Yaskawa INFORM job: ariel_test_28-12.JBI

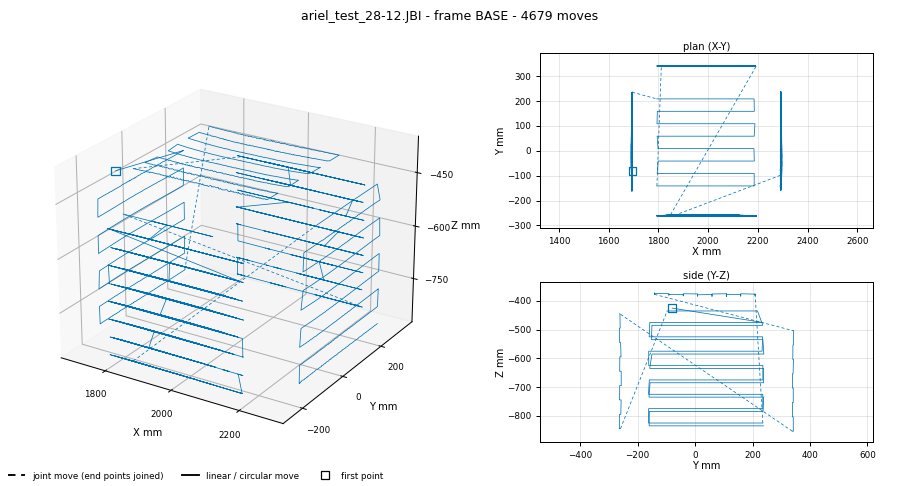
[picture p0: tool path of ariel_test_28-12.JBI in frame BASE, 4679 of 4679 moves have a stored position in this frame; points joined in program order, loops and branches not executed]
/JOB
//NAME ARIEL_TEST
//POS
///NPOS 4679,0,0,0,0,0
///TOOL 0
///POSTYPE BASE
///RECTAN
///RCONF 1,0,0,0,0,0,0,0,0,0,0,0,0,0,0,0,0,0,0,0,0,0,0,0
C00000=1696.132000,-80.047400,-425.128800,-2.796034,72.857313,-92.928025
C00001=1694.988400,235.674100,-475.128800,91.633140,81.554813,1.615741
C00002=1694.763900,232.398000,-475.128800,113.107598,87.891726,23.090199
C00003=1694.793600,228.055300,-475.128800,-70.657155,88.596464,-160.663095
C00004=1695.151200,224.781200,-475.128800,-66.440186,88.699596,-156.446126
C00005=1695.130800,221.009900,-475.128800,-43.934404,88.980346,-133.934614
C00006=1695.054300,219.997000,-475.128800,-8.926682,88.791270,-98.926893
C00007=1695.058500,217.094900,-475.128800,-159.081732,88.567816,110.924629
C00008=1694.887700,215.803300,-475.128800,-11.676880,88.842836,-101.677090
C00009=1695.188800,212.462700,-475.128800,-4.371668,86.453602,-94.377608
C00010=1695.133100,208.131800,-475.128800,-42.633790,89.398605,-132.634000
C00011=1695.189200,206.048000,-475.128800,-13.493156,89.587681,-103.493367
C00012=1695.116300,201.470900,-475.128800,50.191103,88.590734,-39.803378
C00013=1694.965700,197.460000,-475.128800,48.460770,89.272554,-41.539440
C00014=1695.140400,191.185200,-475.128800,17.492401,89.639247,-72.502079
C00015=1694.918000,187.331000,-475.128800,31.885101,88.860024,-58.109380
C00016=1695.110400,184.389700,-475.128800,64.853093,89.364227,-25.147118
C00017=1694.969600,179.240300,-475.128800,-12.100869,87.914644,-102.106809
C00018=1695.056000,175.417900,-475.128800,38.898105,88.590734,-51.090647
C00019=1694.747200,170.987700,-475.128800,47.629982,87.817241,-42.347311
C00020=1694.650000,164.775100,-475.128800,16.432430,88.510520,-73.562051
C00021=1694.533900,162.575300,-475.128800,42.089480,88.390199,-47.899272
C00022=1694.373600,158.045800,-475.128800,56.997841,88.556357,-32.990910
C00023=1695.089100,155.989400,-475.128800,-6.348372,88.344362,-96.354312
C00024=1695.185800,152.477800,-475.128800,-65.809932,88.149557,-155.821602
C00025=1694.724600,149.203700,-475.128800,6.033246,87.261472,-83.961235
C00026=1695.104800,146.728300,-475.128800,19.486295,88.923050,-70.513916
C00027=1694.834300,143.853900,-475.128800,47.733114,88.705326,-42.255637
C00028=1693.934200,141.094100,-475.128800,115.748934,87.490655,25.725805
C00029=1693.799200,137.257000,-475.128800,99.190453,86.671326,9.173054
C00030=1693.895200,133.651800,-475.128800,38.038668,87.828700,-51.938624
C00031=1693.476900,130.746700,-475.128800,21.720830,87.026560,-68.250733
C00032=1694.334900,128.603600,-475.128800,25.382030,86.785917,-64.583803
C00033=1695.164800,125.432200,-475.128800,143.904080,88.711055,53.898140
C00034=1694.863300,121.656100,-475.128800,8.382373,87.026560,-81.606379
C00035=1693.391000,117.740300,-475.128800,20.064982,87.748486,-69.923769
C00036=1694.429700,115.474900,-475.128800,6.205133,87.381793,-83.789348
C00037=1693.264100,112.358400,-475.128800,47.624252,88.350092,-42.364499
C00038=1694.551300,109.480100,-475.128800,-7.053110,87.507844,-97.059050
C00039=1694.104100,106.646300,-475.128800,8.141730,87.198447,-81.847021
C00040=1693.197200,102.981000,-475.128800,-2.950733,87.444819,-92.950943
C00041=1694.004100,100.489400,-475.128800,16.031359,86.929157,-73.951663
C00042=1694.629400,96.503800,-475.128800,0.435448,86.785917,-89.559033
C00043=1693.339800,94.279400,-475.128800,4.153944,86.602571,-85.840537
C00044=1693.243600,89.591100,-475.128800,30.068825,88.395929,-59.919926
C00045=1694.046600,86.533600,-475.128800,-0.435448,87.101044,-90.435658
C00046=1694.079400,83.430500,-475.128800,-14.896903,86.636948,-104.920031
C00047=1694.640600,81.259500,-475.128800,-7.591691,81.062069,-97.683574
C00048=1693.579900,77.591900,-475.128800,-3.701307,86.728621,-93.707247
C00049=1694.579600,74.118800,-475.128800,8.061516,86.677055,-81.927235
C00050=1694.602200,71.620100,-475.128800,5.655093,86.379117,-84.333658
C00051=1693.230300,67.936100,-475.128800,7.574502,86.682785,-82.408520
C00052=1692.692500,63.461100,-475.128800,3.368992,87.301579,-86.625489
C00053=1693.515800,60.204800,-475.128800,-3.540879,86.751540,-93.541090
C00054=1694.397600,57.070500,-475.128800,-1.867842,86.321821,-91.873782
C00055=1695.083600,51.313600,-475.128800,-46.077266,88.854295,-136.083206
C00056=1693.552700,49.260100,-475.128800,3.449206,86.327551,-86.545275
C00057=1693.236600,43.220200,-475.128800,-9.150136,86.361928,-99.167535
C00058=1692.438400,40.123200,-475.128800,-10.250215,86.860402,-100.267614
C00059=1693.005200,36.124700,-475.128800,-0.458366,86.281714,-90.458577
C00060=1694.308400,31.082800,-475.128800,-2.051189,86.493709,-92.057129
C00061=1692.704700,27.503400,-475.128800,2.784575,87.782864,-87.209906
C00062=1693.177400,25.817900,-475.128800,10.880469,87.307309,-79.108283
C00063=1692.952200,22.582800,-475.128800,5.826981,86.052531,-84.161771
C00064=1693.146000,20.159200,-475.128800,3.770062,88.063613,-86.224419
C00065=1694.605100,16.625400,-475.128800,-10.141353,85.754593,-100.170211
C00066=1693.774400,12.699800,-475.128800,-8.978249,86.957805,-98.989918
C00067=1694.221300,10.877900,-475.128800,9.396508,85.456655,-80.569325
C00068=1693.353500,8.692400,-475.128800,-10.588260,87.479196,-100.599930
C00069=1695.395900,6.553600,-475.128800,-14.278108,75.962744,-104.696578
C00070=1694.514400,2.859000,-475.128800,-3.775792,86.293174,-93.781732
C00071=1694.492400,-1.569500,-475.128800,-24.327788,87.284391,-114.356646
C00072=1692.776900,-3.735100,-475.128800,-27.318628,87.261472,-117.347486
C00073=1694.690400,-6.961900,-475.128800,-12.060762,85.788971,-102.089620
C00074=1694.113600,-9.973800,-475.128800,-4.881600,87.410441,-94.887540
C00075=1695.315300,-12.616400,-475.128800,5.523313,88.338633,-84.471168
C00076=1693.186800,-16.477300,-475.128800,-14.810959,86.969264,-104.828358
C00077=1694.776500,-17.860800,-475.128800,-8.147460,86.396306,-98.159129
C00078=1693.169700,-22.210600,-475.128800,-23.491270,87.536492,-113.508669
C00079=1694.236600,-24.585300,-475.128800,-9.763201,86.023883,-99.786330
C00080=1693.849200,-28.361700,-475.128800,-19.784233,87.204176,-109.807361
C00081=1694.081800,-32.852400,-475.128800,-27.788453,87.393252,-117.817311
C00082=1694.169000,-36.280800,-475.128800,-40.880539,87.215636,-130.915127
C00083=1694.436000,-38.893400,-475.128800,-11.493533,86.333281,-101.516662
C00084=1693.377800,-42.844200,-475.128800,-15.429753,87.020830,-105.452882
C00085=1693.729500,-46.013500,-475.128800,-5.689471,87.284391,-95.695411
C00086=1693.512300,-48.882800,-475.128800,-21.319760,87.272931,-111.337159
C00087=1694.121900,-53.479200,-475.128800,-2.097026,87.370334,-92.097236
C00088=1694.254700,-55.606600,-475.128800,-8.663122,87.123962,-98.674791
C00089=1695.480200,-60.498300,-475.128800,-7.551584,88.361551,-97.551794
C00090=1694.880500,-63.263300,-475.128800,-10.066868,86.344740,-100.089997
C00091=1695.519400,-67.371500,-475.128800,-4.279995,86.465061,-94.291664
C00092=1695.154700,-69.634000,-475.128800,-16.690261,86.906238,-106.713389
C00093=1694.837500,-73.212500,-475.128800,-14.346863,87.209906,-104.364262
C00094=1695.406500,-77.363100,-475.128800,-22.505782,86.992182,-112.534641
C00095=1695.106600,-81.047500,-475.128800,-14.696367,88.143827,-104.702307
C00096=1694.416400,-84.097200,-475.128800,-20.317083,87.628165,-110.334483
C00097=1695.519600,-87.829700,-475.128800,82.540300,88.986075,-7.459910
C00098=1694.707800,-90.627800,-475.128800,-9.660068,86.911968,-99.671738
C00099=1695.330000,-93.501100,-475.128800,-21.336948,87.679731,-111.354347
C00100=1695.363400,-99.305300,-475.128800,-13.200948,87.582329,-103.212617
C00101=1694.622800,-103.431100,-475.128800,-32.750268,88.315715,-122.761937
C00102=1695.475000,-107.547000,-475.128800,2.710090,87.840160,-87.290120
C00103=1694.908200,-111.406000,-475.128800,-12.536317,88.235500,-102.542257
C00104=1695.600100,-115.157400,-475.128800,63.403510,89.793946,-26.596701
C00105=1694.895300,-121.393400,-475.128800,-19.469106,88.373010,-109.475046
C00106=1695.267600,-125.384400,-475.128800,-1.890761,88.424577,-91.896701
C00107=1694.736800,-129.294900,-475.128800,-21.904177,89.049101,-111.910117
C00108=1694.843800,-133.799800,-475.128800,-11.694069,88.355822,-101.694279
C00109=1695.271400,-139.102900,-475.128800,-14.432807,88.751162,-104.438747
C00110=1695.095400,-144.244300,-475.128800,-2.475178,88.281337,-92.475388
C00111=1694.850400,-148.261100,-475.128800,-17.985145,88.453224,-107.991085
C00112=1695.327400,-150.030400,-475.128800,46.959621,88.785540,-43.034860
C00113=1695.394800,-153.452400,-475.128800,127.414354,87.192717,37.385496
C00114=1694.805400,-157.684500,-475.128800,-67.276704,86.963534,-157.305563
C00115=1694.500400,-159.876400,-525.128800,-78.924936,82.712187,-169.011090
C00116=1694.421900,-156.702300,-525.128800,-95.036509,88.539168,174.964122
C00117=1694.689000,-153.571800,-525.128800,-16.822041,89.484548,-106.822251
C00118=1694.622100,-150.053500,-525.128800,-18.987821,88.865754,-108.993761
C00119=1694.362400,-147.366300,-525.128800,-40.221637,88.865754,-130.221848
C00120=1694.470800,-144.581100,-525.128800,-53.118917,88.842836,-143.124857
C00121=1694.487200,-142.921900,-525.128800,-69.241950,88.911591,-159.247890
C00122=1694.727000,-138.966100,-525.128800,-58.361481,89.238177,-148.367421
C00123=1694.454100,-135.239700,-525.128800,-40.026832,88.573546,-130.032772
C00124=1694.239400,-130.327700,-525.128800,-74.828288,88.739703,-164.834228
C00125=1694.291700,-126.172900,-525.128800,-35.735378,88.327174,-125.747047
C00126=1693.961600,-120.293700,-525.128800,-44.455795,88.161016,-134.467465
C00127=1694.229600,-117.327700,-525.128800,-39.677327,88.378740,-129.688997
C00128=1693.955300,-112.124600,-525.128800,-39.012696,88.550627,-129.018636
C00129=1694.120500,-109.056600,-525.128800,-37.087558,88.544898,-127.099228
C00130=1693.350900,-104.310500,-525.128800,-49.807221,87.840160,-139.824620
C00131=1693.551400,-100.440500,-525.128800,-37.339660,87.800053,-127.357059
C00132=1693.489700,-95.539000,-525.128800,-61.277836,87.232824,-151.306695
C00133=1693.865700,-92.922100,-525.128800,-39.562736,87.439089,-129.591594
C00134=1693.249200,-88.499300,-525.128800,-41.917592,88.774081,-131.923532
C00135=1693.006200,-86.270900,-525.128800,-63.541019,88.373010,-153.546960
C00136=1693.393100,-79.718400,-525.128800,-36.887023,87.857348,-126.904422
C00137=1693.031700,-76.883500,-525.128800,-29.226577,87.651083,-119.249706
C00138=1693.235600,-73.650000,-525.128800,-33.667000,87.943292,-123.684399
C00139=1692.490700,-67.602900,-525.128800,-23.044363,87.496385,-113.061762
C00140=1693.098200,-63.993300,-525.128800,-33.162797,87.502114,-123.191656
C00141=1692.056100,-60.055400,-525.128800,-46.856488,88.653760,-136.862429
C00142=1692.699200,-57.465500,-525.128800,-34.411845,88.172475,-124.423515
C00143=1692.339800,-53.601900,-525.128800,-27.215495,88.034965,-117.227165
C00144=1692.501500,-49.582900,-525.128800,-18.157033,88.092261,-108.168702
C00145=1691.991300,-47.866600,-525.128800,-46.999728,88.292796,-137.017127
C00146=1692.189200,-44.341200,-525.128800,-17.383540,87.759945,-107.395209
C00147=1691.755300,-40.515100,-525.128800,-28.390059,88.464684,-118.401728
C00148=1692.760800,-37.856600,-525.128800,-26.757129,86.321821,-116.803176
C00149=1692.377400,-34.007100,-525.128800,-22.929771,88.831377,-112.929981
C00150=1692.333500,-29.550300,-525.128800,-22.843827,88.355822,-112.849767
C00151=1691.906200,-26.667400,-525.128800,-25.783101,88.212582,-115.794770
C00152=1692.601600,-23.052500,-525.128800,-46.506984,87.651083,-136.530113
C00153=1691.715700,-19.895400,-525.128800,-46.524173,88.378740,-136.535843
C00154=1691.346100,-17.017200,-525.128800,-23.370948,88.269878,-113.382618
C00155=1691.553100,-15.002600,-525.128800,-34.423304,88.350092,-124.434974
C00156=1691.985700,-9.968700,-525.128800,-10.416373,88.075072,-100.422313
C00157=1691.467400,-6.304400,-525.128800,-5.809792,88.023506,-95.815732
C00158=1691.911100,-3.077000,-525.128800,-20.746802,88.716785,-110.752742
C00159=1691.862600,0.698400,-525.128800,-8.072975,88.052154,-98.078915
C00160=1691.612400,3.808600,-525.128800,-39.127288,89.049101,-129.127498
C00161=1692.269100,7.928600,-525.128800,-24.430920,87.204176,-114.454049
C00162=1691.326600,9.877800,-525.128800,-26.018013,88.928779,-116.023954
C00163=1691.066200,12.948400,-525.128800,-66.268299,87.828700,-156.279968
C00164=1691.291700,15.880200,-525.128800,-9.734553,87.519303,-99.746223
C00165=1691.603000,21.223400,-525.128800,-14.014548,88.659489,-104.020488
C00166=1691.244300,23.875200,-525.128800,20.116548,88.728244,-69.877933
C00167=1691.672000,27.568300,-525.128800,-40.141423,88.258419,-130.153093
C00168=1691.918800,29.995600,-525.128800,-5.030569,87.295850,-95.036509
C00169=1691.532200,34.742900,-525.128800,62.280512,89.272554,-27.713969
C00170=1691.777300,36.968100,-525.128800,1.638659,87.633895,-88.361551
C00171=1692.094100,41.761800,-525.128800,7.465640,88.842836,-82.528841
C00172=1692.187100,44.735300,-525.128800,16.243353,87.937562,-73.745398
C00173=1691.171000,47.416500,-525.128800,33.867535,88.968886,-56.132675
C00174=1691.446100,51.083700,-525.128800,10.582530,88.504791,-79.417680
C00175=1691.301500,52.729200,-525.128800,50.815627,89.163692,-39.178854
C00176=1691.411400,56.907700,-525.128800,101.276020,88.808458,11.270080
C00177=1691.256200,60.771300,-525.128800,20.420216,88.487602,-69.574265
C00178=1691.909500,62.038600,-525.128800,2.807493,88.390199,-87.192717
C00179=1692.124100,67.281200,-525.128800,17.062683,88.350092,-72.931798
C00180=1692.099300,70.838300,-525.128800,26.373247,88.441765,-63.615504
C00181=1692.157500,72.684000,-525.128800,18.649776,88.378740,-71.338975
C00182=1691.565800,76.598500,-525.128800,3.036676,88.464684,-86.963534
C00183=1691.909400,80.224700,-525.128800,105.017434,89.123585,15.017224
C00184=1692.286100,84.108200,-525.128800,18.718531,88.298526,-71.275950
C00185=1691.948700,86.578200,-525.128800,38.038668,88.430306,-51.950083
C00186=1691.934400,90.287100,-525.128800,18.030982,88.607923,-71.963499
C00187=1692.085000,93.239200,-525.128800,42.868702,88.040695,-47.114319
C00188=1692.449200,96.809000,-525.128800,-8.600097,87.565140,-98.611766
C00189=1691.972100,100.726900,-525.128800,51.932895,88.327174,-38.055857
C00190=1692.777100,102.244500,-525.128800,51.503176,87.003641,-38.456927
C00191=1692.585200,107.563200,-525.128800,43.831271,88.052154,-46.151750
C00192=1692.245700,109.667000,-525.128800,90.315337,88.562086,0.315127
C00193=1692.710700,113.138300,-525.128800,77.658700,88.017776,-12.330052
C00194=1692.487800,115.926400,-525.128800,54.436720,88.441765,-35.552031
C00195=1692.585500,119.868600,-525.128800,70.542564,88.550627,-19.451917
C00196=1692.703700,124.136900,-525.128800,68.038738,87.857348,-21.950013
C00197=1693.348100,127.989000,-525.128800,14.123410,89.008993,-75.871071
C00198=1693.014600,131.500300,-525.128800,52.689199,87.960481,-37.293823
C00199=1693.004100,135.286200,-525.128800,69.190383,88.023506,-20.798368
C00200=1693.062300,138.337900,-525.128800,70.296192,88.670948,-19.698289
C00201=1693.695300,142.853900,-525.128800,36.308335,87.164069,-53.657498
C00202=1693.927400,146.038400,-525.128800,25.032526,87.926103,-64.956225
C00203=1693.303900,150.565200,-525.128800,86.190041,88.590734,-3.810169
C00204=1693.469800,156.957300,-525.128800,171.486268,89.662165,81.486058
C00205=1693.614100,160.194900,-525.128800,68.479916,88.057884,-21.508836
C00206=1693.876900,164.625000,-525.128800,83.050232,88.745433,-6.949978
C00207=1694.292400,168.627500,-525.128800,69.012766,88.831377,-20.987444
C00208=1693.978700,172.496500,-525.128800,66.422997,88.390199,-23.565754
C00209=1694.116300,176.139200,-525.128800,93.793191,88.991805,3.792981
C00210=1694.081500,181.483900,-525.128800,58.418777,88.550627,-31.569975
C00211=1694.426900,184.221100,-525.128800,61.741932,88.648030,-28.252549
C00212=1694.402500,190.301700,-525.128800,32.217417,89.008993,-57.777064
C00213=1694.649600,195.955200,-525.128800,59.765228,88.722515,-30.229253
C00214=1694.804700,197.877500,-525.128800,52.637633,89.026182,-37.356848
C00215=1694.710300,202.217900,-525.128800,65.454699,89.324120,-24.545512
C00216=1694.828100,206.371000,-525.128800,47.612793,89.014723,-42.381688
C00217=1694.680600,209.763000,-525.128800,130.336439,88.579275,40.324770
C00218=1694.784900,212.216100,-525.128800,55.021137,88.917320,-34.979073
C00219=1694.849000,214.324600,-525.128800,1.747521,87.880267,-88.252689
C00220=1694.724400,215.988100,-525.128800,31.403817,88.481872,-58.584935
C00221=1694.889400,219.187200,-525.128800,4.898789,88.745433,-85.101421
C00222=1694.788600,221.768000,-525.128800,-122.830692,84.247714,147.301720
C00223=1694.756300,224.941700,-525.128800,-136.604598,88.269878,133.407493
C00224=1694.729100,227.663700,-525.128800,7.081758,89.822594,-82.918452
C00225=1694.687300,230.259700,-525.128800,50.511959,89.135044,-39.488251
C00226=1694.723200,234.923700,-525.128800,92.355067,83.353900,2.337668
C00227=1694.806300,233.203100,-575.128800,103.653795,82.620514,13.544722
C00228=1694.742300,231.059300,-575.128800,75.120497,86.952075,-14.862525
C00229=1694.693700,226.262900,-575.128800,-78.369167,89.008993,-168.369378
C00230=1694.887000,224.564300,-575.128800,-9.866333,89.862701,-99.866544
C00231=1694.695600,221.286200,-575.128800,-22.906853,89.478819,-112.907063
C00232=1694.713100,219.344300,-575.128800,73.464648,89.387146,-16.535562
C00233=1694.584600,216.524100,-575.128800,139.297499,89.725191,49.297289
C00234=1694.630300,213.463400,-575.128800,27.129552,88.968886,-62.870659
C00235=1694.668100,210.962700,-575.128800,162.061112,88.728244,72.055172
C00236=1694.607400,208.721700,-575.128800,108.357778,89.049101,18.357568
C00237=1694.629100,206.423000,-575.128800,24.935123,89.094937,-65.065087
C00238=1694.628700,202.253300,-575.128800,69.952417,89.220988,-20.042064
C00239=1694.515400,199.405300,-575.128800,104.089243,89.112126,14.083303
C00240=1694.346400,194.510600,-575.128800,53.239238,88.791270,-36.755243
C00241=1694.248400,188.122200,-575.128800,78.437922,88.527709,-11.556559
C00242=1694.228200,183.278500,-575.128800,96.904352,88.224041,6.904141
C00243=1693.970700,179.423000,-575.128800,78.953584,88.218312,-11.040897
C00244=1693.868200,172.668500,-575.128800,53.353830,88.579275,-36.640651
C00245=1693.812400,169.950500,-575.128800,112.523181,88.367281,22.517241
C00246=1693.709200,166.789600,-575.128800,79.956260,89.106396,-10.038221
C00247=1693.646200,162.728400,-575.128800,71.470755,88.212582,-18.517996
C00248=1693.661500,159.420200,-575.128800,85.055585,88.206853,-4.938896
C00249=1693.425500,155.227500,-575.128800,91.696166,88.034965,1.695955
C00250=1693.320300,151.517000,-575.128800,78.861911,88.648030,-11.132570
C00251=1693.201800,147.367900,-575.128800,74.587646,88.390199,-15.406835
C00252=1692.996500,142.122500,-575.128800,106.043029,87.496385,16.031359
C00253=1692.897500,140.572100,-575.128800,57.874467,88.109450,-32.114284
C00254=1692.852900,136.432100,-575.128800,102.232859,86.997912,12.215460
C00255=1692.607500,133.096600,-575.128800,108.311942,88.166746,18.300272
C00256=1692.506800,127.929600,-575.128800,84.007072,88.097991,-5.987409
C00257=1692.637100,126.345400,-575.128800,103.814223,88.487602,13.808283
C00258=1692.460100,120.405100,-575.128800,121.426946,87.891726,31.409546
C00259=1692.265600,116.228300,-575.128800,86.465061,88.636571,-3.535150
C00260=1692.250600,112.447400,-575.128800,102.278696,88.510520,12.272756
C00261=1692.136600,109.594700,-575.128800,72.055172,88.413117,-17.933579
C00262=1691.893000,104.059400,-575.128800,56.694174,88.476143,-33.294577
C00263=1691.813200,101.461400,-575.128800,106.782144,88.636571,16.781934
C00264=1691.820100,97.498400,-575.128800,48.300342,88.716785,-41.694139
C00265=1691.695000,93.109800,-575.128800,97.007484,88.642300,7.007274
C00266=1691.744500,90.048900,-575.128800,96.686628,88.670948,6.686417
C00267=1691.683500,85.860600,-575.128800,134.988857,88.602193,44.982916
C00268=1691.585900,83.286900,-575.128800,85.640002,89.364227,-4.360209
C00269=1691.337700,79.352400,-575.128800,57.043678,88.728244,-32.950803
C00270=1691.369100,74.414100,-575.128800,75.424164,89.255365,-14.576046
C00271=1691.218900,72.542400,-575.128800,119.862771,89.610599,29.862560
C00272=1691.295600,67.757100,-575.128800,66.852716,89.106396,-23.147495
C00273=1691.304300,64.282100,-575.128800,163.579451,87.828700,73.567781
C00274=1691.097900,62.191800,-575.128800,56.992112,89.152233,-33.002369
C00275=1690.987500,56.823900,-575.128800,-140.225691,89.284013,129.774941
C00276=1691.165600,55.524500,-575.128800,34.383197,88.367281,-55.605554
C00277=1691.027500,51.901500,-575.128800,118.229841,89.725191,28.229631
C00278=1690.928900,47.456300,-575.128800,56.241537,88.653760,-33.747214
C00279=1690.984000,45.810200,-575.128800,-8.462587,88.298526,-98.468527
C00280=1691.087500,41.819000,-575.128800,-52.030297,89.146503,-142.036237
C00281=1691.043600,39.213400,-575.128800,142.305528,89.513196,52.305317
C00282=1691.026500,35.327600,-575.128800,-28.487462,89.564763,-118.487672
C00283=1690.873600,32.032400,-575.128800,45.848083,89.180881,-44.152128
C00284=1690.821200,30.213600,-575.128800,33.913372,88.161016,-56.069650
C00285=1690.929400,26.425500,-575.128800,-12.662367,88.613653,-102.668307
C00286=1690.815600,23.772000,-575.128800,-111.904387,89.335579,158.096244
C00287=1690.808600,19.852900,-575.128800,57.759875,89.610599,-32.240335
C00288=1690.950900,16.612700,-575.128800,-115.525480,89.856971,154.475151
C00289=1690.737500,11.905700,-575.128800,-109.039598,88.894402,160.966763
C00290=1690.920900,8.527600,-575.128800,-84.270633,89.026182,-174.270843
C00291=1690.739300,5.954200,-575.128800,167.045845,89.885619,77.045635
C00292=1690.841100,2.739900,-575.128800,-19.812881,89.627788,-109.813091
C00293=1690.672400,-1.372900,-575.128800,31.770510,89.581951,-58.229701
C00294=1690.806600,-3.662500,-575.128800,-41.470685,88.464684,-131.476625
C00295=1691.056800,-8.688600,-575.128800,-28.029095,89.049101,-118.029306
C00296=1690.987500,-12.668800,-575.128800,6.514530,88.814188,-83.485680
C00297=1690.795700,-20.036900,-575.128800,-41.344634,89.432982,-131.344845
C00298=1690.997900,-24.547800,-575.128800,-76.890936,89.049101,-166.896876
C00299=1690.918100,-30.269200,-575.128800,-25.966447,89.135044,-115.972387
C00300=1691.294200,-35.152800,-575.128800,-25.296087,88.224041,-115.302027
C00301=1691.022000,-39.070400,-575.128800,-46.294990,89.037641,-136.300930
C00302=1691.086400,-41.699200,-575.128800,-46.799193,88.762622,-136.805133
C00303=1691.265600,-47.309800,-575.128800,-46.346556,88.848565,-136.352496
C00304=1691.355200,-50.600100,-575.128800,-19.864447,88.991805,-109.864657
C00305=1691.892600,-55.259700,-575.128800,-41.751435,88.075072,-131.763104
C00306=1691.475100,-59.480400,-575.128800,-78.111336,88.178205,-168.117276
C00307=1691.274300,-63.897400,-575.128800,-78.472300,88.212582,-168.478240
C00308=1691.851500,-66.924200,-575.128800,-38.823620,87.966210,-128.841019
C00309=1691.543400,-71.041500,-575.128800,-128.193577,87.800053,141.829973
C00310=1691.724300,-73.351300,-575.128800,-3.111161,88.029236,-93.111371
C00311=1692.211900,-78.850500,-575.128800,-89.123585,88.877213,-179.123795
C00312=1692.125800,-79.622100,-575.128800,-76.782074,88.837106,-166.788014
C00313=1692.001400,-84.001300,-575.128800,-76.438299,88.648030,-166.438510
C00314=1692.577700,-87.866400,-575.128800,-56.258726,88.825647,-146.258936
C00315=1692.045800,-91.980500,-575.128800,-95.620926,88.579275,174.379705
C00316=1692.173600,-94.043900,-575.128800,-85.508221,87.777134,-175.508432
C00317=1692.553100,-100.118900,-575.128800,-73.298491,88.109450,-163.304431
C00318=1692.848000,-103.049700,-575.128800,-65.809932,88.143827,-155.821602
C00319=1693.065100,-107.930200,-575.128800,-76.151821,87.513574,-166.163490
C00320=1692.948700,-112.113100,-575.128800,-59.564692,88.733974,-149.570632
C00321=1693.011800,-116.306100,-575.128800,-82.815320,88.000588,-172.815530
C00322=1693.309500,-121.879900,-575.128800,-72.765640,87.055207,-162.788769
C00323=1693.330000,-125.985400,-575.128800,-81.228227,87.410441,-171.234167
C00324=1693.636700,-128.998600,-575.128800,-81.950153,88.052154,-171.950364
C00325=1693.762900,-132.765600,-575.128800,-79.560919,88.304255,-169.566859
C00326=1693.867800,-137.386300,-575.128800,-126.560647,88.648030,143.445714
C00327=1694.041100,-140.149600,-575.128800,-69.791989,88.069343,-159.803659
C00328=1694.038600,-142.787500,-575.128800,-94.813056,88.057884,175.187575
C00329=1694.000600,-144.618300,-575.128800,-71.533781,87.966210,-161.545450
C00330=1694.203100,-147.692000,-575.128800,-95.334448,88.573546,174.666184
C00331=1694.311200,-152.225200,-575.128800,-102.175564,89.255365,167.825068
C00332=1694.376400,-154.259400,-575.128800,31.060042,89.719461,-58.940168
C00333=1694.414700,-156.252300,-575.128800,-114.247784,87.341686,155.775765
C00334=1694.517600,-158.357200,-575.128800,-103.183969,88.888672,166.822392
C00335=1694.945200,-161.433200,-575.128800,-94.738571,78.260305,175.359463
C00336=1694.553400,-161.479100,-625.128800,-68.806502,79.050987,-159.156216
C00337=1694.756200,-158.430600,-625.128800,-76.220575,83.760700,-166.301000
C00338=1694.559700,-156.743200,-625.128800,-104.387181,86.413495,165.636369
C00339=1694.303200,-153.567800,-625.128800,-61.564315,87.559410,-151.587444
C00340=1694.320200,-150.343100,-625.128800,-84.299280,87.450548,-174.299491
C00341=1693.989800,-147.719700,-625.128800,-78.013933,86.992182,-168.031333
C00342=1693.810300,-142.914800,-625.128800,-75.481460,87.101044,-165.498859
C00343=1693.818300,-139.261400,-625.128800,-95.110994,87.370334,174.895367
C00344=1693.699800,-134.943000,-625.128800,-92.120154,88.023506,177.880477
C00345=1693.573700,-130.480400,-625.128800,-96.119400,87.645354,173.886961
C00346=1693.153700,-126.406300,-625.128800,-86.946345,87.123962,-176.952285
C00347=1693.106600,-121.856200,-625.128800,-78.718671,87.095314,-168.730341
C00348=1692.960600,-118.089600,-625.128800,-84.133123,87.926103,-174.139063
C00349=1692.713100,-112.713100,-625.128800,-82.248091,87.971940,-172.254032
C00350=1692.412300,-110.341100,-625.128800,-74.702237,88.246960,-164.708177
C00351=1692.432900,-106.464300,-625.128800,-76.358085,88.212582,-166.364025
C00352=1692.347100,-102.865600,-625.128800,-97.574713,88.046424,172.431648
C00353=1692.024000,-98.807000,-625.128800,-67.660586,87.725568,-157.677985
C00354=1692.063300,-93.005100,-625.128800,-73.859989,88.860024,-163.860200
C00355=1692.032700,-88.429400,-625.128800,-83.353900,87.954751,-173.354110
C00356=1691.922900,-85.154300,-625.128800,-81.577731,87.897455,-171.583671
C00357=1691.639900,-80.293400,-625.128800,-118.332973,88.103720,151.679117
C00358=1691.561900,-76.884200,-625.128800,-63.225893,88.499061,-153.237562
C00359=1691.419600,-71.985100,-625.128800,-22.769343,86.459331,-112.809660
C00360=1691.352000,-67.828900,-625.128800,-54.316399,88.796999,-144.322339
C00361=1691.103500,-64.509200,-625.128800,-48.231587,88.373010,-138.237527
C00362=1691.180500,-61.617600,-625.128800,-24.001202,88.997534,-114.001412
C00363=1691.089200,-57.626000,-625.128800,-73.819882,88.928779,-163.820093
C00364=1691.159300,-54.104900,-625.128800,151.656199,89.925726,61.655988
C00365=1691.154800,-50.557900,-625.128800,-38.674651,89.020453,-128.674862
C00366=1691.026100,-48.692300,-625.128800,-45.722032,88.665219,-135.727972
C00367=1690.951200,-44.611100,-625.128800,-74.421488,89.014723,-164.421698
C00368=1690.795700,-42.130000,-625.128800,-39.333553,88.957427,-129.333763
C00369=1690.759500,-37.278500,-625.128800,-49.532201,89.467360,-139.532412
C00370=1690.847700,-34.944000,-625.128800,-94.371878,89.369957,175.628753
C00371=1690.742800,-31.427000,-625.128800,-121.129007,89.455901,148.871624
C00372=1690.778000,-28.339400,-625.128800,-12.278486,89.020453,-102.278696
C00373=1690.609300,-25.061600,-625.128800,40.049750,89.748109,-49.944731
C00374=1690.613800,-21.692600,-625.128800,124.732912,89.043371,34.726972
C00375=1690.768600,-19.120600,-625.128800,-153.718847,88.756892,116.287514
C00376=1690.638900,-13.464400,-625.128800,-174.746398,89.031912,95.254233
C00377=1690.663300,-8.718300,-625.128800,151.908300,89.536115,61.908090
C00378=1690.737200,-6.140600,-625.128800,-21.663534,89.352768,-111.663745
C00379=1690.630500,-4.212800,-625.128800,-49.566579,89.324120,-139.566789
C00380=1690.744500,-0.158000,-625.128800,-167.389620,88.934509,102.611012
C00381=1690.633000,2.934700,-625.128800,54.889357,88.900131,-35.105124
C00382=1690.812700,6.829400,-625.128800,19.423269,89.444441,-70.576941
C00383=1690.813200,11.135600,-625.128800,109.589637,89.484548,19.589427
C00384=1690.874600,15.819000,-625.128800,-149.209669,89.450171,120.796692
C00385=1691.095200,20.063900,-625.128800,104.009029,88.017776,14.003089
C00386=1690.840000,22.530800,-625.128800,95.655304,89.329850,5.655093
C00387=1690.961700,26.623700,-625.128800,68.869527,88.791270,-21.124954
C00388=1690.939700,30.121100,-625.128800,56.751470,89.392875,-33.248741
C00389=1690.878700,33.744200,-625.128800,40.215908,88.923050,-49.784303
C00390=1690.938300,36.801700,-625.128800,175.405299,89.496008,85.405089
C00391=1690.897900,40.528300,-625.128800,-120.212275,89.897078,149.782627
C00392=1691.261800,42.787500,-625.128800,84.958182,88.882943,-5.042029
C00393=1691.064500,46.432900,-625.128800,75.653347,89.312661,-14.341134
C00394=1691.059900,50.483700,-625.128800,168.718882,88.882943,78.718671
C00395=1691.194500,54.245900,-625.128800,115.216083,88.814188,25.215873
C00396=1691.318200,58.791200,-625.128800,99.247749,89.140774,9.247539
C00397=1691.361100,61.495100,-625.128800,88.281337,88.344362,-1.718873
C00398=1691.203500,66.319200,-625.128800,136.707730,88.481872,46.696060
C00399=1691.260000,69.455700,-625.128800,-114.064438,89.473089,155.936194
C00400=1691.776200,71.904900,-625.128800,122.280653,89.289743,32.274713
C00401=1691.544400,76.312700,-625.128800,138.587031,88.057884,48.575362
C00402=1691.652800,79.136800,-625.128800,143.669167,88.195393,53.657498
C00403=1691.489400,81.695000,-625.128800,24.705940,88.779810,-65.288541
C00404=1691.825400,84.982900,-625.128800,86.728621,88.464684,-3.271589
C00405=1691.761600,87.171800,-625.128800,83.027314,88.550627,-6.972896
C00406=1691.764200,91.864500,-625.128800,125.248574,88.550627,35.236904
C00407=1691.811400,95.976400,-625.128800,111.285593,87.949022,21.273923
C00408=1692.051200,97.972400,-625.128800,81.915776,88.917320,-8.078705
C00409=1692.046000,101.259300,-625.128800,54.740388,87.805782,-35.242634
C00410=1692.323400,105.961800,-625.128800,131.602676,88.573546,41.596736
C00411=1692.101100,108.639200,-625.128800,117.582399,88.470413,27.576459
C00412=1692.376400,112.436100,-625.128800,114.391024,87.393252,24.373625
C00413=1692.334200,115.215700,-625.128800,93.352014,87.908915,3.351803
C00414=1692.524500,118.458000,-625.128800,89.392875,88.980346,-0.607335
C00415=1692.672300,121.812200,-625.128800,85.193095,88.728244,-4.807116
C00416=1692.830200,126.268000,-625.128800,118.722585,88.544898,28.716645
C00417=1692.865100,130.574200,-625.128800,142.609195,88.854295,52.603255
C00418=1693.032000,134.375000,-625.128800,98.422690,88.281337,8.416750
C00419=1692.945200,136.693300,-625.128800,128.829560,87.834430,38.806431
C00420=1693.180800,141.376200,-625.128800,45.481390,88.252689,-44.501632
C00421=1692.988800,143.518500,-625.128800,17.876283,88.344362,-72.112468
C00422=1693.249900,148.889500,-625.128800,46.581469,88.344362,-43.407283
C00423=1693.385400,151.667000,-625.128800,24.110064,88.590734,-65.884417
C00424=1693.535700,156.208600,-625.128800,77.991015,88.304255,-12.003466
C00425=1693.629400,160.429000,-625.128800,100.078538,88.636571,10.072598
C00426=1693.584500,162.586800,-625.128800,79.715618,88.688137,-10.278863
C00427=1693.916300,167.276800,-625.128800,-126.377301,88.888672,143.629060
C00428=1693.851100,170.854900,-625.128800,82.534570,88.430306,-7.459910
C00429=1694.063000,174.582000,-625.128800,120.326867,88.499061,30.315197
C00430=1693.968600,177.425700,-625.128800,66.033386,89.089208,-23.966825
C00431=1694.060600,181.015300,-625.128800,61.673177,88.957427,-28.321304
C00432=1694.049400,183.667700,-625.128800,81.904317,88.688137,-8.090164
C00433=1694.155500,186.522300,-625.128800,58.699526,87.937562,-31.283496
C00434=1694.273000,190.850700,-625.128800,64.331701,89.507467,-25.668509
C00435=1694.261300,194.576800,-625.128800,80.557866,88.825647,-9.436615
C00436=1694.375000,196.487000,-625.128800,75.699184,88.733974,-14.301027
C00437=1694.430400,199.264100,-625.128800,114.843660,88.573546,24.837720
C00438=1694.342900,202.564500,-625.128800,41.447767,89.690813,-48.552444
C00439=1694.471500,206.831100,-625.128800,54.734658,89.175151,-35.259823
C00440=1694.648000,209.887000,-625.128800,-95.494876,89.776757,174.505756
C00441=1694.667400,213.074200,-625.128800,94.560955,88.819917,4.560744
C00442=1694.646900,215.930400,-625.128800,158.342616,89.077748,68.342406
C00443=1694.487900,218.634100,-625.128800,130.101527,89.421523,40.095587
C00444=1694.698800,222.258500,-625.128800,139.692840,88.413117,49.686900
C00445=1694.679900,225.429200,-625.128800,173.038984,89.031912,83.033044
C00446=1694.702200,227.521500,-625.128800,-120.739396,88.206853,149.272694
C00447=1694.633200,230.367900,-625.128800,84.683162,89.261095,-5.317048
C00448=1694.651000,232.143900,-625.128800,89.324120,87.519303,-0.676090
C00449=1694.803700,234.775100,-625.128800,94.503659,78.203009,4.411775
C00450=1695.065800,235.983200,-625.128800,95.151101,74.329815,4.956085
C00451=1695.245600,235.879800,-675.128800,93.564008,73.481837,3.420558
C00452=1694.638500,231.558800,-675.128800,126.892963,88.860024,36.887023
C00453=1694.621900,230.657600,-675.128800,145.239071,89.014723,55.238861
C00454=1694.786200,227.972500,-675.128800,116.402106,89.238177,26.396166
C00455=1694.835000,225.201500,-675.128800,-99.471203,89.925726,170.529429
C00456=1694.776100,222.095400,-675.128800,108.311942,88.894402,18.306002
C00457=1694.564200,216.891900,-675.128800,75.447082,88.384469,-14.547398
C00458=1694.567000,212.845800,-675.128800,70.238896,89.381416,-19.761314
C00459=1694.574200,210.852200,-675.128800,73.338598,89.157963,-16.661613
C00460=1694.586900,206.438900,-675.128800,119.438782,88.447495,29.427112
C00461=1694.540200,204.609800,-675.128800,117.605317,88.940239,27.605107
C00462=1694.307000,199.817500,-675.128800,93.655681,88.321444,3.655471
C00463=1694.179800,195.707200,-675.128800,89.243906,89.031912,-0.756304
C00464=1694.211100,192.151100,-675.128800,67.334000,89.358498,-22.666210
C00465=1694.109000,188.180000,-675.128800,92.784785,88.424577,2.784575
C00466=1694.138300,183.661700,-675.128800,82.614784,89.599140,-7.385426
C00467=1694.048700,180.823800,-675.128800,73.149522,88.854295,-16.844959
C00468=1693.896800,177.478100,-675.128800,87.553681,88.378740,-2.446530
C00469=1694.085000,174.820600,-675.128800,132.146986,88.625112,42.141046
C00470=1693.776500,169.386000,-675.128800,98.508634,88.493331,8.502694
C00471=1693.704000,165.885600,-675.128800,106.604527,88.585005,16.598587
C00472=1693.611600,162.289200,-675.128800,116.298973,89.026182,26.293033
C00473=1693.880400,157.966100,-675.128800,134.839888,89.335579,44.839677
C00474=1693.699500,154.392400,-675.128800,106.764956,89.335579,16.764745
C00475=1693.583400,150.822700,-675.128800,43.802623,89.622058,-46.197587
C00476=1693.439800,147.709800,-675.128800,114.797824,89.014723,24.797613
C00477=1693.225500,145.601300,-675.128800,149.633658,88.436036,59.627718
C00478=1693.427300,142.311000,-675.128800,78.346249,88.401658,-11.653962
C00479=1693.079400,137.686600,-675.128800,110.792849,88.688137,20.786909
C00480=1692.987800,136.923000,-675.128800,71.980688,89.616329,-18.013793
C00481=1693.339100,131.791500,-675.128800,114.425401,88.373010,24.419461
C00482=1693.013200,129.588700,-675.128800,141.847161,89.438712,51.846951
C00483=1692.767800,125.654500,-675.128800,104.604905,88.722515,14.598965
C00484=1692.813500,122.006800,-675.128800,102.101079,87.857348,12.089409
C00485=1692.812400,119.181400,-675.128800,110.993384,89.100667,20.987444
C00486=1692.816300,114.880900,-675.128800,134.284118,88.470413,44.272449
C00487=1692.599800,111.705200,-675.128800,145.645872,89.478819,55.645661
C00488=1692.551400,105.915500,-675.128800,138.856322,88.917320,48.850382
C00489=1692.353700,103.666500,-675.128800,141.617978,88.642300,51.606309
C00490=1692.606100,99.889700,-675.128800,136.386874,89.157963,46.380934
C00491=1692.461400,95.053800,-675.128800,117.840230,89.157963,27.840019
C00492=1692.235600,91.643900,-675.128800,101.132780,87.817241,11.121111
C00493=1692.499100,87.954600,-675.128800,153.821979,87.639624,63.804580
C00494=1692.535700,86.109600,-675.128800,80.065122,89.008993,-9.935088
C00495=1692.496300,81.933500,-675.128800,179.914477,88.103720,89.914267
C00496=1691.996100,77.963500,-675.128800,105.458612,88.808458,15.458401
C00497=1692.115300,72.851200,-675.128800,93.924971,89.215258,3.924761
C00498=1692.245000,70.999500,-675.128800,151.404097,87.633895,61.386698
C00499=1691.752200,66.406500,-675.128800,102.765710,88.648030,12.765500
C00500=1692.183700,63.371500,-675.128800,124.068281,88.533439,34.062341
C00501=1691.637500,59.884500,-675.128800,62.022681,88.745433,-27.971800
C00502=1691.839500,57.285200,-675.128800,133.791375,88.103720,43.779705
C00503=1691.528000,53.894600,-675.128800,103.470448,89.014723,13.470238
C00504=1691.820800,47.982200,-675.128800,110.603773,89.220988,20.603562
C00505=1691.923300,45.596500,-675.128800,135.223769,87.880267,45.206370
C00506=1691.279200,41.081500,-675.128800,129.179064,88.235500,39.167395
C00507=1691.624800,35.574800,-675.128800,142.695139,89.003264,52.689199
C00508=1691.600200,33.164300,-675.128800,136.736378,88.779810,46.724708
C00509=1690.980500,26.763900,-675.128800,-18.558103,89.427253,-108.558313
C00510=1690.949800,21.099300,-675.128800,107.572826,88.825647,17.566886
C00511=1691.143900,16.194100,-675.128800,116.167193,89.066289,26.166983
C00512=1691.424200,11.751000,-675.128800,133.756997,89.249636,43.756787
C00513=1691.094100,7.273500,-675.128800,110.483452,88.218312,20.471782
C00514=1690.870700,3.199800,-675.128800,150.418610,89.656436,60.418399
C00515=1690.954700,-1.233400,-675.128800,141.709651,89.043371,51.709441
C00516=1690.851200,-6.282800,-675.128800,113.331052,88.968886,23.325112
C00517=1691.009100,-8.317700,-675.128800,107.905142,89.381416,17.904931
C00518=1690.981900,-12.509000,-675.128800,140.878863,88.831377,50.872923
C00519=1690.792300,-14.250200,-675.128800,121.753531,88.544898,31.747591
C00520=1690.997600,-19.700400,-675.128800,130.141634,88.407388,40.129964
C00521=1690.764000,-22.287900,-675.128800,-165.624910,89.198070,104.375722
C00522=1690.559100,-24.595400,-675.128800,81.858480,89.415794,-8.136001
C00523=1690.630200,-27.426600,-675.128800,-4.108107,89.719461,-94.108318
C00524=1690.758100,-32.489900,-675.128800,-74.581916,89.822594,-164.582127
C00525=1690.754300,-34.883200,-675.128800,175.686049,89.329850,85.685838
C00526=1690.749700,-39.937000,-675.128800,-48.432122,89.799675,-138.432333
C00527=1690.725000,-44.414800,-675.128800,-132.794428,89.415794,137.206203
C00528=1690.788800,-47.195600,-675.128800,-58.625042,89.306932,-148.625252
C00529=1690.761600,-51.141700,-675.128800,-113.944117,89.094937,156.056515
C00530=1690.857400,-54.909700,-675.128800,-31.461113,89.484548,-121.461323
C00531=1690.932400,-56.457700,-675.128800,-104.014758,89.238177,165.991603
C00532=1690.952900,-62.657800,-675.128800,-60.469966,89.616329,-150.470176
C00533=1690.945300,-67.080200,-675.128800,-115.817689,89.289743,154.182943
C00534=1690.993000,-68.922200,-675.128800,-120.321137,88.865754,149.685224
C00535=1691.168300,-74.266900,-675.128800,-71.361893,89.387146,-161.362104
C00536=1691.235600,-77.564600,-675.128800,18.168492,89.123585,-71.831719
C00537=1691.168700,-79.420700,-675.128800,-70.376406,89.347039,-160.376616
C00538=1691.279200,-83.136400,-675.128800,-6.222322,89.243906,-96.222532
C00539=1691.188200,-86.832400,-675.128800,-86.974993,89.112126,-176.975204
C00540=1691.324500,-92.414000,-675.128800,-80.775590,88.819917,-170.775800
C00541=1691.540900,-98.964500,-675.128800,-86.860402,88.092261,-176.860612
C00542=1691.811800,-105.062900,-675.128800,-83.193472,87.989129,-173.199412
C00543=1692.210800,-112.360100,-675.128800,-63.323296,87.800053,-153.340695
C00544=1692.209800,-115.189500,-675.128800,-93.117101,88.241230,176.883531
C00545=1692.266600,-119.780500,-675.128800,-77.796209,87.060937,-167.813609
C00546=1692.437600,-123.193100,-675.128800,-84.912345,87.439089,-174.918285
C00547=1692.778300,-128.012500,-675.128800,-71.046767,87.341686,-161.064166
C00548=1692.792700,-133.918000,-675.128800,-85.926481,87.570869,-175.926691
C00549=1693.046700,-136.595400,-675.128800,-101.608335,86.963534,168.409485
C00550=1693.198600,-140.397200,-675.128800,-75.114767,86.946345,-165.132166
C00551=1693.224100,-144.578100,-675.128800,-64.228569,88.097991,-154.245968
C00552=1693.395600,-149.262600,-675.128800,-70.468079,87.232824,-160.491208
C00553=1693.731500,-154.414400,-675.128800,-70.370676,88.441765,-160.376616
C00554=1694.180800,-157.429500,-675.128800,-79.721348,85.955128,-169.744476
C00555=1694.113900,-159.350400,-675.128800,-80.832886,84.327928,-170.878933
C00556=1693.613400,-162.296700,-725.128800,-77.292007,71.866096,-167.905282
C00557=1693.452700,-158.027000,-725.128800,-75.126226,87.106774,-165.143625
C00558=1693.478500,-154.036400,-725.128800,-82.047556,88.693867,-172.047767
C00559=1693.526000,-153.060000,-725.128800,-98.267991,87.599517,171.738370
C00560=1693.283000,-149.465700,-725.128800,-97.534605,86.717162,172.477485
C00561=1693.196900,-145.572300,-725.128800,-107.429587,88.046424,162.582504
C00562=1693.175300,-142.266200,-725.128800,-88.670948,87.708379,-178.671159
C00563=1692.987800,-139.610700,-725.128800,-87.370334,87.106774,-177.376274
C00564=1692.683800,-134.034900,-725.128800,-81.663675,88.470413,-171.669615
C00565=1692.547500,-129.592900,-725.128800,-74.295437,87.822971,-164.307107
C00566=1692.553100,-124.530400,-725.128800,-103.659524,88.149557,166.352566
C00567=1692.491800,-118.202100,-725.128800,-105.578933,86.591112,164.450346
C00568=1692.058500,-113.505000,-725.128800,-95.231315,87.966210,174.769316
C00569=1692.024000,-110.890100,-725.128800,-92.624357,88.504791,177.376274
C00570=1691.717300,-106.496400,-725.128800,-94.045292,88.516250,175.955339
C00571=1691.849400,-102.992300,-725.128800,-124.406326,87.771405,145.611494
C00572=1691.820500,-99.398600,-725.128800,-120.550320,88.407388,149.461770
C00573=1691.518300,-93.894700,-725.128800,-95.185479,88.751162,174.815153
C00574=1691.727100,-90.920000,-725.128800,-136.157690,88.865754,133.848671
C00575=1691.521400,-88.468300,-725.128800,-137.544248,89.667895,132.456383
C00576=1691.558700,-83.592800,-725.128800,-117.204247,89.043371,152.796385
C00577=1691.757700,-81.533600,-725.128800,-152.905247,88.464684,117.101114
C00578=1691.409200,-75.937500,-725.128800,-107.200403,89.616329,162.800228
C00579=1691.267200,-73.868600,-725.128800,-135.750890,89.398605,134.249741
C00580=1691.368100,-69.992100,-725.128800,-139.847539,88.481872,130.158822
C00581=1691.497000,-66.905600,-725.128800,-153.816250,88.521979,116.195841
C00582=1691.202900,-62.642000,-725.128800,79.354655,89.742379,-10.639826
C00583=1690.949100,-58.842500,-725.128800,-81.703782,89.811134,-171.703992
C00584=1691.102500,-55.456000,-725.128800,-67.511617,89.713732,-157.511827
C00585=1691.059900,-52.475800,-725.128800,67.311082,89.908537,-22.689129
C00586=1691.516900,-46.324700,-725.128800,-173.967175,89.100667,96.033456
C00587=1691.447900,-42.499900,-725.128800,-170.907581,88.814188,99.093051
C00588=1691.440200,-37.363600,-725.128800,165.630639,88.819917,75.624699
C00589=1691.264200,-34.202600,-725.128800,171.068009,89.049101,81.067798
C00590=1691.613100,-29.953700,-725.128800,147.026700,88.579275,57.020760
C00591=1691.398400,-25.866100,-725.128800,167.916741,88.625112,77.910801
C00592=1691.470200,-22.076100,-725.128800,149.221128,88.258419,59.209459
C00593=1691.500500,-18.159800,-725.128800,-177.599728,89.249636,92.400904
C00594=1691.331100,-12.737700,-725.128800,129.081662,89.152233,39.081451
C00595=1691.544800,-7.886200,-725.128800,95.712600,88.854295,5.712389
C00596=1691.477900,-4.905400,-725.128800,155.271562,88.562086,65.265622
C00597=1691.865100,-1.307700,-725.128800,31.283496,87.691191,-58.693797
C00598=1691.572300,1.972800,-725.128800,125.941853,89.473089,35.941642
C00599=1691.649200,6.374200,-725.128800,69.946688,89.369957,-20.053523
C00600=1691.423100,10.417600,-725.128800,175.405299,89.054830,85.405089
C00601=1691.470900,15.426900,-725.128800,179.249846,88.103720,89.249636
C00602=1691.943200,16.520100,-725.128800,117.868878,88.080802,27.857208
C00603=1692.137300,20.796100,-725.128800,127.729481,88.579275,37.717812
C00604=1691.889800,23.766900,-725.128800,111.652286,88.384469,21.640616
C00605=1692.127200,26.966200,-725.128800,146.218829,88.693867,56.212889
C00606=1692.577900,31.210600,-725.128800,128.170659,88.940239,38.164719
C00607=1692.179100,36.844000,-725.128800,161.407940,88.963157,71.407730
C00608=1692.102800,39.325100,-725.128800,154.314723,89.301202,64.314513
C00609=1691.963000,43.711500,-725.128800,86.161393,88.499061,-3.838817
C00610=1692.276500,46.641800,-725.128800,130.061419,88.493331,40.049750
C00611=1692.298200,50.614000,-725.128800,150.367044,87.800053,60.349645
C00612=1692.932000,53.849400,-725.128800,150.619145,88.865754,60.618935
C00613=1692.972100,58.007400,-725.128800,162.651259,87.645354,72.639589
C00614=1692.852200,64.094100,-725.128800,136.936913,88.246960,46.919514
C00615=1692.938300,66.408700,-725.128800,132.238659,88.401658,42.226990
C00616=1693.033100,71.877200,-725.128800,147.313179,89.140774,57.312968
C00617=1692.911800,73.086300,-725.128800,155.586689,87.989129,65.569290
C00618=1692.580300,77.916200,-725.128800,88.688137,88.395929,-1.312073
C00619=1693.081500,80.440600,-725.128800,148.797139,88.625112,58.785470
C00620=1692.999600,84.182900,-725.128800,141.698192,88.304255,51.680793
C00621=1693.143900,88.816500,-725.128800,138.833403,88.865754,48.827463
C00622=1692.709600,92.833400,-725.128800,142.786812,89.089208,52.780872
C00623=1692.909300,96.351400,-725.128800,157.592042,88.739703,67.586102
C00624=1693.248800,98.029200,-725.128800,125.775695,88.304255,35.764026
C00625=1692.980800,102.527300,-725.128800,150.206616,88.418847,60.200676
C00626=1693.040000,105.070900,-725.128800,141.193989,88.556357,51.182320
C00627=1693.018400,109.244300,-725.128800,124.985013,88.751162,34.973344
C00628=1693.458600,111.504500,-725.128800,142.351364,88.458954,52.339695
C00629=1693.230000,117.177600,-725.128800,126.692428,88.367281,36.680758
C00630=1693.513000,120.828700,-725.128800,149.817004,89.570492,59.816794
C00631=1693.238500,126.613700,-725.128800,115.708827,89.094937,25.702887
C00632=1693.802000,128.159300,-725.128800,118.292866,89.673625,28.292656
C00633=1693.445700,132.606700,-725.128800,80.809967,88.464684,-9.184513
C00634=1693.419900,137.271300,-725.128800,81.096446,88.613653,-8.903764
C00635=1693.877200,140.934900,-725.128800,128.915504,89.054830,38.909564
C00636=1693.696700,145.465800,-725.128800,94.721383,88.642300,4.721172
C00637=1693.975900,148.239900,-725.128800,159.901061,88.848565,69.895121
C00638=1694.009000,152.974400,-725.128800,112.591936,89.037641,22.591726
C00639=1693.924900,156.030400,-725.128800,167.888093,89.438712,77.887883
C00640=1693.898900,160.064500,-725.128800,114.104545,89.438712,24.104334
C00641=1694.022600,163.945000,-725.128800,122.504106,88.252689,32.492437
C00642=1694.158500,168.032600,-725.128800,75.160604,88.825647,-14.833877
C00643=1694.079700,171.275500,-725.128800,6.915601,89.043371,-83.084610
C00644=1694.151900,176.630100,-725.128800,149.095077,89.518926,59.094867
C00645=1694.067500,178.046700,-725.128800,23.204791,88.527709,-66.783961
C00646=1694.156400,183.068400,-725.128800,95.242774,88.831377,5.242564
C00647=1694.232100,186.390400,-725.128800,110.328753,88.768351,20.322813
C00648=1694.315000,189.126700,-725.128800,74.856936,88.630841,-15.137545
C00649=1694.536000,192.256500,-725.128800,100.874949,88.808458,10.874739
C00650=1694.451600,196.132200,-725.128800,110.867333,89.329850,20.867123
C00651=1694.330700,199.616800,-725.128800,165.160814,88.779810,75.154874
C00652=1694.507800,203.227000,-725.128800,118.281407,89.060560,28.281197
C00653=1694.640600,208.150100,-725.128800,131.018259,89.043371,41.012319
C00654=1694.478800,210.745400,-725.128800,101.184347,88.848565,11.184136
C00655=1694.662500,216.049300,-725.128800,35.723919,89.570492,-54.276292
C00656=1694.674000,217.352300,-725.128800,107.716065,88.768351,17.715855
C00657=1694.625200,221.604500,-725.128800,94.010915,87.719838,4.010705
C00658=1694.737600,223.176500,-725.128800,91.083101,88.556357,1.082890
C00659=1694.916500,226.335600,-725.128800,-175.485513,89.501737,94.515118
C00660=1694.902300,227.683700,-725.128800,78.684294,89.220988,-11.310187
C00661=1694.903500,231.089500,-725.128800,43.264043,89.180881,-46.736167
C00662=1694.957700,234.305800,-725.128800,89.215258,83.239308,-0.779223
C00663=1695.307700,235.674100,-725.128800,83.886751,78.569702,-5.993139
C00664=1695.280500,235.559200,-775.128800,91.025805,73.562051,0.985487
C00665=1695.159900,234.589200,-775.128800,96.938729,81.319900,6.858305
C00666=1694.773400,231.875000,-775.128800,85.049855,86.453602,-4.944626
C00667=1694.791500,229.585100,-775.128800,101.705738,88.126638,11.699798
C00668=1694.805900,225.869400,-775.128800,-15.727691,88.762622,-105.733632
C00669=1694.794300,223.920100,-775.128800,21.674993,89.644977,-68.325217
C00670=1694.786500,222.595300,-775.128800,-155.649715,89.060560,114.356646
C00671=1694.646800,218.486500,-775.128800,91.673247,89.163692,1.673037
C00672=1694.643700,215.167800,-775.128800,30.830859,88.539168,-59.163622
C00673=1694.783500,210.666400,-775.128800,81.910046,88.968886,-8.090164
C00674=1694.659000,207.861600,-775.128800,129.488462,88.636571,39.482522
C00675=1694.726600,204.677000,-775.128800,-96.635062,89.742379,173.365570
C00676=1694.675100,201.200900,-775.128800,162.456453,89.513196,72.456243
C00677=1694.820400,199.708000,-775.128800,58.911520,88.802729,-31.082960
C00678=1694.695600,195.486900,-775.128800,122.658805,89.753839,32.658594
C00679=1694.396100,191.453900,-775.128800,178.184145,89.478819,88.183934
C00680=1694.646100,189.710100,-775.128800,154.979354,88.533439,64.973414
C00681=1694.371100,185.227200,-775.128800,96.405879,88.860024,6.405668
C00682=1694.384000,183.786000,-775.128800,112.190866,89.198070,22.184926
C00683=1694.617200,180.852500,-775.128800,-45.945486,89.576222,-135.945696
C00684=1694.318500,176.831800,-775.128800,-147.273072,88.716785,122.739019
C00685=1694.484800,171.631000,-775.128800,179.994691,89.438712,89.994481
C00686=1694.549900,170.698200,-775.128800,-170.540888,89.467360,99.459744
C00687=1694.315400,166.804000,-775.128800,-25.066904,89.450171,-115.067114
C00688=1694.518200,164.098000,-775.128800,-36.629192,89.788216,-126.629402
C00689=1694.521000,160.609400,-775.128800,-46.535632,88.699596,-136.541572
C00690=1694.399400,158.024200,-775.128800,128.485786,89.094937,38.485575
C00691=1694.100000,155.305900,-775.128800,-166.873958,89.604870,103.126674
C00692=1694.580300,150.859200,-775.128800,177.725778,88.877213,87.725568
C00693=1694.108700,146.701800,-775.128800,28.773940,89.324120,-61.220540
C00694=1694.275300,144.221200,-775.128800,8.611556,89.243906,-81.388655
C00695=1694.161300,140.123800,-775.128800,-172.276950,89.730920,97.723682
C00696=1694.260600,135.787900,-775.128800,178.631052,89.043371,88.630841
C00697=1694.433900,132.332000,-775.128800,177.937773,89.054830,87.937562
C00698=1694.373200,129.758300,-775.128800,-93.048346,89.369957,176.952285
C00699=1694.474300,125.985300,-775.128800,-143.703545,87.679731,126.320005
C00700=1694.650000,123.183500,-775.128800,-143.480091,87.949022,126.537729
C00701=1694.005200,118.931700,-775.128800,90.103343,89.295472,0.103132
C00702=1694.023300,115.371200,-775.128800,162.765850,88.888672,72.765640
C00703=1694.243000,111.268900,-775.128800,151.392638,88.894402,61.386698
C00704=1694.349500,107.562900,-775.128800,155.987760,89.599140,65.987549
C00705=1693.895700,105.422300,-775.128800,146.258936,89.461630,56.258726
C00706=1694.008300,100.769400,-775.128800,163.247135,89.014723,73.246925
C00707=1693.806100,96.840000,-775.128800,72.032254,89.753839,-17.967956
C00708=1694.008300,93.264500,-775.128800,150.212345,88.235500,60.200676
C00709=1693.666400,89.449200,-775.128800,158.778064,89.478819,68.777854
C00710=1694.240400,85.928500,-775.128800,142.649302,88.458954,52.637633
C00711=1693.879900,81.183800,-775.128800,136.719189,88.882943,46.713249
C00712=1693.933400,78.390900,-775.128800,-176.786128,89.289743,93.214504
C00713=1694.247700,74.843500,-775.128800,158.164999,88.178205,68.159059
C00714=1693.474700,71.802200,-775.128800,167.292217,86.894779,77.274818
C00715=1693.254000,68.307700,-775.128800,139.996508,89.639247,49.996297
C00716=1693.596300,64.411600,-775.128800,118.900202,87.398982,28.877073
C00717=1693.292400,62.160200,-775.128800,162.038194,86.281714,72.003606
C00718=1694.049800,58.527700,-775.128800,-179.851452,87.341686,90.149179
C00719=1693.009700,56.555000,-775.128800,132.290225,89.175151,42.284285
C00720=1693.085300,51.786400,-775.128800,153.621444,88.464684,63.615504
C00721=1693.390000,48.460800,-775.128800,159.477073,89.215258,69.476862
C00722=1693.441200,45.567400,-775.128800,124.108388,88.413117,34.096718
C00723=1692.734400,41.255200,-775.128800,138.409415,86.929157,48.369097
C00724=1693.264500,40.032600,-775.128800,127.259656,88.539168,37.253716
C00725=1692.977800,36.970700,-775.128800,150.768114,88.304255,60.756445
C00726=1693.785200,31.002200,-775.128800,164.570667,88.653760,74.564727
C00727=1693.321000,29.063000,-775.128800,89.748109,89.008993,-0.252101
C00728=1693.681900,25.546800,-775.128800,154.194402,88.040695,64.177003
C00729=1693.703700,21.608200,-775.128800,143.531657,88.206853,53.514258
C00730=1692.607800,17.413000,-775.128800,124.887611,89.473089,34.887400
C00731=1692.705800,13.934000,-775.128800,148.464824,88.281337,58.453154
C00732=1692.582400,10.554800,-775.128800,121.552996,88.579275,31.547056
C00733=1693.159600,6.119500,-775.128800,159.964087,89.112126,69.963876
C00734=1692.987100,2.306600,-775.128800,153.730306,87.920374,63.712907
C00735=1693.198300,-0.580000,-775.128800,134.731026,89.020453,44.725085
C00736=1693.262400,-3.471300,-775.128800,134.295578,89.942915,44.295367
C00737=1692.884100,-7.851100,-775.128800,148.762762,87.851619,58.739633
C00738=1692.399400,-12.054200,-775.128800,171.291462,88.670948,81.291252
C00739=1692.613800,-14.656500,-775.128800,106.959761,88.539168,16.953821
C00740=1692.178400,-17.963200,-775.128800,176.396516,88.138098,86.396306
C00741=1692.992300,-22.676100,-775.128800,-179.295683,87.479196,90.704949
C00742=1693.367300,-24.450800,-775.128800,-14.742204,86.551005,-104.765333
C00743=1692.140100,-28.211700,-775.128800,136.747837,88.802729,46.741897
C00744=1691.974200,-32.842600,-775.128800,128.290980,88.596464,38.285040
C00745=1691.865800,-34.678400,-775.128800,142.809730,88.395929,52.803790
C00746=1693.154000,-38.635300,-775.128800,102.628200,88.470413,12.627990
C00747=1692.169000,-41.325200,-775.128800,-166.747907,87.805782,103.258454
C00748=1691.840700,-47.021000,-775.128800,170.506510,88.321444,80.500570
C00749=1691.929200,-50.154500,-775.128800,178.774291,88.905861,88.774081
C00750=1692.398400,-53.005600,-775.128800,-175.284978,88.258419,94.715653
C00751=1693.146700,-56.114400,-775.128800,169.916364,88.097991,79.910424
C00752=1692.493900,-59.588500,-775.128800,154.245968,88.023506,64.234298
C00753=1692.138700,-63.237200,-775.128800,-173.869773,88.693867,96.130859
C00754=1692.114600,-66.379500,-775.128800,-177.960691,88.395929,92.039940
C00755=1692.843800,-69.024500,-775.128800,161.001140,89.381416,71.000930
C00756=1691.957500,-73.917600,-775.128800,173.571834,89.163692,83.571624
C00757=1691.814200,-76.987200,-775.128800,168.930876,89.427253,78.930666
C00758=1692.733700,-80.165700,-775.128800,-174.522944,88.596464,95.477687
C00759=1692.780000,-84.946900,-775.128800,-154.538177,88.630841,115.468184
C00760=1692.187500,-88.466200,-775.128800,-132.886101,89.381416,137.120260
C00761=1692.254400,-91.320700,-775.128800,-165.561884,88.945968,104.438747
C00762=1692.211200,-96.461400,-775.128800,175.697508,88.092261,85.691568
C00763=1692.013900,-98.631000,-775.128800,-110.517829,89.369957,159.482802
C00764=1692.456600,-102.953700,-775.128800,-173.073361,88.413117,96.933000
C00765=1692.753900,-105.142600,-775.128800,-171.566482,87.822971,98.439879
C00766=1692.791500,-109.369100,-775.128800,-163.579451,89.398605,106.421181
C00767=1692.367700,-113.387800,-775.128800,-146.619900,89.392875,123.380732
C00768=1692.802000,-116.780100,-775.128800,-134.444547,88.831377,135.561814
C00769=1692.428300,-120.154800,-775.128800,-70.674344,88.682408,-160.674554
C00770=1692.995400,-123.926200,-775.128800,-134.484654,88.120909,135.533166
C00771=1692.710300,-127.569900,-775.128800,-108.598420,88.166746,161.407940
C00772=1692.717600,-131.204100,-775.128800,-83.416925,88.189664,-173.422865
C00773=1693.137600,-134.656200,-775.128800,-169.566859,87.868807,100.439501
C00774=1692.815700,-138.280300,-775.128800,-133.115285,88.877213,136.891076
C00775=1693.104900,-143.140200,-775.128800,-117.313109,87.633895,152.704712
C00776=1693.340500,-146.610200,-775.128800,-153.140159,88.453224,116.871931
C00777=1693.161700,-150.894800,-775.128800,-81.102176,88.722515,-171.102386
C00778=1693.309100,-152.742400,-775.128800,-108.111406,88.516250,161.894955
C00779=1693.292700,-156.731700,-775.128800,88.052154,87.295850,-1.948057
C00780=1693.053300,-159.441300,-775.128800,17.068413,87.502114,-72.920339
C00781=1693.169700,-161.869700,-775.128800,-81.640756,81.491787,-171.732640
C00782=1694.095100,-162.262300,-825.128800,-78.758779,80.620891,-168.907958
C00783=1693.815100,-161.320100,-825.128800,-91.111749,84.133123,178.894612
C00784=1693.694300,-159.411200,-825.128800,-74.347003,84.774835,-164.410239
C00785=1693.835100,-155.897300,-825.128800,81.342818,88.115179,-8.651663
C00786=1693.900600,-152.136400,-825.128800,-65.471887,89.467360,-155.472098
C00787=1693.454100,-149.528600,-825.128800,7.116136,89.306932,-82.884075
C00788=1693.684300,-147.537400,-825.128800,-146.430824,89.432982,123.569808
C00789=1693.724600,-142.723600,-825.128800,167.847986,88.659489,77.847776
C00790=1693.435600,-138.200500,-825.128800,-139.910564,88.418847,130.101527
C00791=1693.263800,-134.290800,-825.128800,-141.577871,88.968886,128.422760
C00792=1693.940700,-128.596300,-825.128800,-152.813574,88.579275,117.192787
C00793=1694.179400,-124.135700,-825.128800,178.631052,89.295472,88.630841
C00794=1694.185000,-120.565700,-825.128800,0.664631,87.227095,-89.329850
C00795=1693.074200,-118.342600,-825.128800,-128.772264,88.453224,141.234096
C00796=1693.871000,-114.604000,-825.128800,0.928192,72.903150,-89.026182
C00797=1693.048400,-112.378000,-825.128800,172.334246,88.424577,82.334035
C00798=1694.316100,-109.326900,-825.128800,10.679933,86.826024,-79.308818
C00799=1693.190300,-106.315300,-825.128800,-159.797929,88.246960,110.208432
C00800=1693.523100,-102.267200,-825.128800,-173.445784,88.407388,96.560577
C00801=1693.270400,-98.307700,-825.128800,170.741423,87.926103,80.735483
C00802=1693.937200,-94.548100,-825.128800,166.003062,87.152610,75.985663
C00803=1693.556200,-92.849400,-825.128800,155.162700,88.562086,65.156760
C00804=1694.360300,-89.471700,-825.128800,-5.362885,88.332903,-95.363095
C00805=1693.850400,-84.352600,-825.128800,177.972150,87.599517,87.971940
C00806=1693.997500,-80.760300,-825.128800,-178.327384,87.049478,91.673247
C00807=1694.146000,-75.961900,-825.128800,144.562981,86.900509,54.528393
C00808=1694.179800,-75.053100,-825.128800,164.817039,87.651083,74.805370
C00809=1693.313300,-72.193500,-825.128800,173.520268,88.733974,83.520058
C00810=1692.731200,-67.375500,-825.128800,151.106159,88.029236,61.094490
C00811=1693.090200,-63.308200,-825.128800,169.188707,87.593788,79.182767
C00812=1693.444000,-58.799300,-825.128800,-179.839993,88.298526,90.160639
C00813=1694.003400,-56.443800,-825.128800,152.905247,87.588058,62.882118
C00814=1694.156100,-51.698400,-825.128800,178.911801,88.155286,88.905861
C00815=1693.179100,-48.358500,-825.128800,-136.386874,87.845889,133.630947
C00816=1694.877900,-45.134800,-825.128800,28.836966,86.487979,-61.117408
C00817=1694.494200,-43.968200,-825.128800,1.787628,78.248846,-88.178205
C00818=1694.827400,-39.536300,-825.128800,39.041344,89.501737,-50.958866
C00819=1694.546400,-38.068900,-825.128800,146.018294,85.863455,55.949329
C00820=1694.047000,-34.851100,-825.128800,144.488497,88.012047,54.476827
C00821=1693.287500,-32.741600,-825.128800,143.182153,87.857348,53.164754
C00822=1693.637400,-28.246900,-825.128800,-156.738334,87.049478,113.285215
C00823=1694.872000,-25.166400,-825.128800,23.829315,87.186988,-66.142248
C00824=1694.206600,-19.961900,-825.128800,160.451101,87.714109,70.433702
C00825=1693.988100,-16.926300,-825.128800,166.249434,87.416171,76.232035
C00826=1695.007900,-10.270700,-825.128800,135.172203,89.432982,45.171993
C00827=1693.494500,-9.092000,-825.128800,129.975476,89.610599,39.975265
C00828=1693.831900,-4.675700,-825.128800,152.143213,87.181258,62.114355
C00829=1693.821100,-0.716500,-825.128800,147.318908,88.189664,57.307239
C00830=1695.030200,4.742900,-825.128800,-174.053119,87.416171,95.953242
C00831=1694.269000,8.958500,-825.128800,162.645529,89.129315,72.645319
C00832=1694.252300,12.685000,-825.128800,70.290462,88.309985,-19.698289
C00833=1695.239400,15.959300,-825.128800,25.192954,89.169422,-64.807256
C00834=1694.405600,20.175200,-825.128800,169.910634,89.043371,79.910424
C00835=1695.082500,24.566100,-825.128800,-3.603905,85.347793,-93.615574
C00836=1694.148400,28.214800,-825.128800,163.728420,88.825647,73.722479
C00837=1694.455500,31.493100,-825.128800,174.196358,86.963534,84.190418
C00838=1694.982100,36.164800,-825.128800,165.114977,88.012047,75.103308
C00839=1695.288500,39.974300,-825.128800,111.148083,89.690813,21.147872
C00840=1694.277400,43.704300,-825.128800,145.279179,88.905861,55.273238
C00841=1695.018700,45.352100,-825.128800,156.182565,87.565140,66.165166
C00842=1694.905500,50.154800,-825.128800,151.438475,87.106774,61.409616
C00843=1694.322000,51.954300,-825.128800,164.771203,88.161016,74.759533
C00844=1695.248100,55.346600,-825.128800,136.650434,89.690813,46.650224
C00845=1694.732200,60.073000,-825.128800,148.745573,89.135044,58.739633
C00846=1695.004100,65.468500,-825.128800,-146.745950,87.857348,123.271870
C00847=1694.372900,68.729800,-825.128800,177.645564,88.481872,87.645354
C00848=1694.675100,72.104900,-825.128800,166.702070,88.103720,76.696130
C00849=1695.361000,75.107300,-825.128800,-1.695955,85.330604,-91.701895
C00850=1695.030600,79.516600,-825.128800,171.205519,89.220988,81.205308
C00851=1695.249800,83.262900,-825.128800,-5.672282,79.744266,-95.764166
C00852=1695.418500,86.450900,-825.128800,129.717645,88.395929,39.705975
C00853=1694.684500,90.238400,-825.128800,153.896464,87.891726,63.879065
C00854=1694.504800,92.614200,-825.128800,153.071405,88.865754,63.065465
C00855=1694.979700,96.882900,-825.128800,-166.043169,88.636571,103.957462
C00856=1695.282200,99.955900,-825.128800,-148.310125,86.682785,121.730613
C00857=1694.821800,103.587100,-825.128800,-169.801772,89.364227,100.198859
C00858=1694.415000,106.340500,-825.128800,149.054970,88.413117,59.043301
C00859=1695.139700,109.931800,-825.128800,-173.623401,88.269878,96.377231
C00860=1694.795000,113.963700,-825.128800,160.943845,88.413117,70.937905
C00861=1694.714100,116.480000,-825.128800,154.841844,89.135044,64.841634
C00862=1694.885200,120.619600,-825.128800,-18.214328,89.140774,-108.220268
C00863=1694.939600,125.359200,-825.128800,-165.934307,88.481872,104.066324
C00864=1694.925000,127.362000,-825.128800,165.475941,88.493331,75.470001
C00865=1695.358900,131.443700,-825.128800,-10.170001,84.757647,-100.210318
C00866=1694.821100,135.115200,-825.128800,-151.610362,89.163692,118.390269
C00867=1694.874400,136.578100,-825.128800,-178.321655,88.733974,91.678977
C00868=1694.817300,140.672400,-825.128800,-102.192752,88.739703,167.807879
C00869=1694.890800,145.148600,-825.128800,148.487742,88.974616,58.481802
C00870=1694.568400,148.641200,-825.128800,176.362139,88.785540,86.361928
C00871=1694.859100,151.520700,-825.128800,113.394077,89.507467,23.393867
C00872=1694.992900,157.338400,-825.128800,132.788699,89.662165,42.788488
C00873=1694.959800,162.037500,-825.128800,-77.269088,89.175151,-167.269299
C00874=1694.902300,165.267300,-825.128800,-178.533649,88.951698,91.466982
C00875=1694.742300,172.042500,-825.128800,-175.279249,88.888672,94.721383
C00876=1695.262700,176.077000,-825.128800,173.262437,89.324120,83.256497
C00877=1694.944500,178.401100,-825.128800,168.873581,89.066289,78.873370
C00878=1694.964000,182.387300,-825.128800,174.225006,89.031912,84.219066
C00879=1695.235900,185.808000,-825.128800,125.918935,89.484548,35.918724
C00880=1695.185300,189.761800,-825.128800,-2.177240,89.261095,-92.177450
C00881=1694.829800,192.133500,-825.128800,-12.467562,89.553303,-102.467772
C00882=1694.887300,196.365300,-825.128800,155.111134,88.768351,65.105194
C00883=1694.857400,198.669500,-825.128800,156.778441,89.387146,66.778231
C00884=1694.754900,201.884100,-825.128800,-55.324805,89.650706,-145.325015
C00885=1694.760500,206.123400,-825.128800,-104.656471,89.576222,165.344161
C00886=1694.964400,209.550100,-825.128800,-148.642441,88.934509,121.358191
C00887=1694.769500,213.173500,-825.128800,-133.963262,88.000588,136.054558
C00888=1694.791300,216.621200,-825.128800,20.019145,89.312661,-69.981065
C00889=1695.249100,221.438800,-825.128800,-45.756410,87.341686,-135.785268
C00890=1694.882100,222.542700,-825.128800,-156.033596,87.874537,113.984224
C00891=1695.078800,225.878300,-825.128800,-2.618417,86.390576,-92.624357
C00892=1694.924400,227.268800,-825.128800,174.769316,87.542222,84.763376
C00893=1694.725600,231.410500,-825.128800,84.459709,87.009371,-5.534772
C00894=1694.952900,233.477700,-825.128800,94.927647,84.098745,4.904519
C00895=1695.024000,235.696700,-825.128800,91.856594,76.037229,1.804817
C00896=1793.675300,208.803900,-377.180700,-3.976327,1.157375,-90.000210
C00897=1799.260300,208.803900,-377.522700,-4.417505,-4.572203,-90.000210
C00898=1800.380100,208.803900,-377.828400,-2.887707,0.103132,-90.000210
C00899=1804.392900,208.803900,-377.686800,-2.228806,-4.526367,-90.000210
C00900=1805.238500,208.803900,-377.860100,1.610011,-3.512231,-90.000210
C00901=1809.448600,208.803900,-378.127900,-0.670361,-2.383504,-90.000210
C00902=1810.104200,208.803900,-378.034500,0.389611,-1.128727,-90.000210
C00903=1815.541900,208.803900,-378.409000,-2.320479,-3.506502,-90.000210
C00904=1816.234300,208.803900,-377.866300,-5.523313,1.019865,-90.000210
C00905=1819.888600,208.803900,-378.043200,-2.326209,-2.142862,-90.000210
C00906=1822.893700,208.803900,-378.295700,-9.499640,2.108485,-90.000210
C00907=1825.029800,208.803900,-378.253700,-5.213916,-2.601228,-90.000210
C00908=1828.890100,208.803900,-378.517000,0.802141,-4.079460,-90.000210
C00909=1829.853900,208.803900,-378.619700,-4.956085,1.237589,-90.000210
C00910=1834.434100,208.803900,-378.454300,-0.567228,1.713144,-90.000210
C00911=1835.867300,208.803900,-378.912400,-0.773493,-3.248671,-90.000210
C00912=1839.483600,208.803900,-378.247300,-0.870896,1.140186,-90.000210
C00913=1841.644600,208.803900,-379.037700,-3.838817,-1.942327,-90.000210
C00914=1844.398700,208.803900,-379.133000,-3.151268,-2.584040,-90.000210
C00915=1849.534100,208.803900,-378.682500,-2.011082,-2.108485,-90.000210
C00916=1850.191300,208.803900,-379.604800,-1.575634,-4.073730,-90.000210
C00917=1854.259800,208.803900,-378.938100,2.486637,-2.761657,-90.000210
C00918=1855.552200,208.803900,-378.611200,-6.520260,1.455313,-90.000210
C00919=1859.933400,208.803900,-378.736900,0.475555,-0.040107,-90.000210
C00920=1861.222300,208.803900,-378.901500,0.338045,-1.999623,-90.000210
C00921=1865.407800,208.803900,-379.478700,-0.194806,-1.472502,-90.000210
C00922=1869.854700,208.803900,-378.445000,-1.953786,-2.119944,-90.000210
C00923=1870.486800,208.803900,-378.774100,-6.904141,1.695955,-90.000210
C00924=1874.480400,208.803900,-380.418600,-0.532851,-2.274642,-90.000210
C00925=1875.328200,208.803900,-379.048600,-5.603527,-0.309397,-90.000210
C00926=1879.654100,208.803900,-379.098900,-8.090164,1.816276,-90.000210
C00927=1880.591300,208.803900,-380.274800,-7.121865,-0.647442,-90.000210
C00928=1884.581900,208.803900,-380.691900,-5.637905,-3.122620,-90.000210
C00929=1888.675200,208.803900,-379.466300,0.893814,-1.386558,-90.000210
C00930=1889.688000,208.803900,-379.350200,-3.271589,0.521392,-90.000210
C00931=1893.936000,208.803900,-380.386900,-3.323155,-2.773116,-90.000210
C00932=1894.825000,208.803900,-379.595200,-1.432394,1.002676,-90.000210
C00933=1899.785700,208.803900,-380.090700,-3.386181,0.922462,-90.000210
C00934=1900.882400,208.803900,-380.488800,-3.924761,-1.810547,-90.000210
C00935=1904.672200,208.803900,-379.458500,-4.870141,-2.624147,-90.000210
C00936=1906.870600,208.803900,-381.091800,-3.225752,-1.718873,-90.000210
C00937=1909.764100,208.803900,-380.616900,-3.729955,0.813600,-90.000210
C00938=1915.067100,208.803900,-379.839900,-3.500772,-1.260507,-90.000210
C00939=1915.511400,208.803900,-381.230100,-1.776169,-2.847600,-90.000210
C00940=1919.150500,208.803900,-378.820100,-6.806739,1.346451,-90.000210
C00941=1921.049200,208.803900,-380.439600,-3.368992,-2.303290,-90.000210
C00942=1924.399500,208.803900,-378.784500,-4.182592,-1.094349,-90.000210
C00943=1926.037100,208.803900,-380.778200,-1.610011,-0.269290,-90.000210
C00944=1929.785000,208.803900,-379.554500,-7.545854,0.991217,-90.000210
C00945=1932.448600,208.803900,-380.390500,-5.454558,1.976704,-90.000210
C00946=1934.473700,208.803900,-378.545700,-10.800254,2.715820,-90.000210
C00947=1938.665100,208.803900,-379.236700,-0.716197,1.117268,-90.000210
C00948=1939.972300,208.803900,-381.396100,0.372423,1.787628,-90.000210
C00949=1944.120800,208.803900,-380.121800,-1.214671,-1.758980,-90.000210
C00950=1945.329900,208.803900,-379.766700,-3.638282,-1.472502,-90.000210
C00951=1949.489500,208.803900,-380.873200,-4.629499,2.652795,-90.000210
C00952=1950.750900,208.803900,-379.083500,-4.251347,1.466772,-90.000210
C00953=1954.631300,208.803900,-379.256600,-2.836141,-0.630254,-90.000210
C00954=1956.191500,208.803900,-379.552900,-6.457234,1.329262,-90.000210
C00955=1960.229500,208.803900,-379.116700,-4.721172,-0.790682,-90.000210
C00956=1963.802800,208.803900,-381.137400,-3.374721,-1.145916,-90.000210
C00957=1964.943200,208.803900,-378.752900,-4.050812,-0.292208,-90.000210
C00958=1968.916700,208.803900,-380.754400,-8.336536,1.409476,-90.000210
C00959=1970.139600,208.803900,-380.852600,-3.237212,5.351426,-90.000210
C00960=1973.999800,208.803900,-380.062400,-4.555014,2.990840,-90.000210
C00961=1975.489000,208.803900,-380.490800,-5.867088,-1.042783,-90.000210
C00962=1979.540300,208.803900,-380.741000,-2.217347,2.750197,-90.000210
C00963=1980.841200,208.803900,-379.906700,-2.939273,1.426665,-90.000210
C00964=1984.548200,208.803900,-379.531600,-2.457989,3.896113,-90.000210
C00965=1985.330500,208.803900,-377.747500,-8.909494,5.099324,-90.000210
C00966=1989.044700,208.803900,-380.605200,-1.128727,2.383504,-90.000210
C00967=1990.266000,208.803900,-377.667700,-12.599342,-2.177240,-90.000210
C00968=1994.859100,208.803900,-379.373700,-0.733386,2.079837,-90.000210
C00969=1995.564500,208.803900,-380.385900,-1.776169,-2.681442,-90.000210
C00970=2000.220600,208.803900,-379.669600,-3.924761,1.157375,-90.000210
C00971=2002.199400,208.803900,-379.938700,-3.409099,4.073730,-90.000210
C00972=2005.140200,208.803900,-379.479100,-0.624524,1.695955,-90.000210
C00973=2008.461600,208.803900,-378.774400,-3.248671,4.915978,-90.000210
C00974=2010.347600,208.803900,-379.928800,-5.592068,1.472502,-90.000210
C00975=2014.097700,208.803900,-380.402000,-0.647442,-4.142485,-90.000210
C00976=2014.950600,208.803900,-379.359500,-6.377020,2.979381,-90.000210
C00977=2018.830000,208.803900,-379.797500,-2.778845,-0.343775,-90.000210
C00978=2019.895500,208.803900,-379.005300,-2.950733,-1.117268,-90.000210
C00979=2023.913800,208.803900,-379.490400,0.045837,3.529420,-90.000210
C00980=2024.936800,208.803900,-377.505100,-0.572958,1.535527,-90.000210
C00981=2029.433300,208.803900,-379.336300,-2.280372,-0.189076,-90.000210
C00982=2030.638500,208.803900,-379.630300,-3.013758,0.658901,-90.000210
C00983=2035.518100,208.803900,-379.299100,-2.188699,0.395341,-90.000210
C00984=2036.993600,208.803900,-379.866000,-1.804817,-0.246372,-90.000210
C00985=2040.274600,208.803900,-379.622600,-6.583285,1.037054,-90.000210
C00986=2041.009000,208.803900,-380.443800,-3.569527,1.810547,-90.000210
C00987=2044.440700,208.803900,-379.299400,-7.935465,2.836141,-90.000210
C00988=2049.189800,208.803900,-378.984300,-1.426665,1.501149,-90.000210
C00989=2050.196200,208.803900,-379.315100,-3.781521,1.827735,-90.000210
C00990=2054.969900,208.803900,-377.751700,-2.744468,0.773493,-90.000210
C00991=2056.023600,208.803900,-380.655600,-4.938896,1.077161,-90.000210
C00992=2059.833200,208.803900,-378.961800,-0.355234,-2.715820,-90.000210
C00993=2060.654800,208.803900,-379.561400,-5.317048,-1.850654,-90.000210
C00994=2064.797100,208.803900,-378.210900,-6.554637,0.773493,-90.000210
C00995=2067.348900,208.803900,-379.260100,-4.864412,2.435071,-90.000210
C00996=2070.116900,208.803900,-379.228400,-5.036299,0.710468,-90.000210
C00997=2074.491600,208.803900,-378.624200,-1.856383,0.945380,-90.000210
C00998=2075.255700,208.803900,-379.646200,-2.309020,-1.707414,-90.000210
C00999=2079.276500,208.803900,-379.165700,-1.867842,6.325454,-90.000210
C01000=2079.869400,208.803900,-377.136600,0.286479,3.317426,-90.000210
C01001=2084.185300,208.803900,-378.837700,-6.548908,6.589015,-90.000210
C01002=2085.181600,208.803900,-377.092700,-15.114627,-4.503448,-90.000210
C01003=2088.476400,208.803900,-378.541800,-0.509932,-2.652795,-90.000210
C01004=2090.558700,208.803900,-378.454900,-0.813600,-1.461042,-90.000210
C01005=2094.855400,208.803900,-378.434900,-1.976704,2.509555,-90.000210
C01006=2095.498000,208.803900,-377.348000,-5.042029,2.773116,-90.000210
C01007=2099.183700,208.803900,-377.018700,-5.013381,9.075651,-90.000210
C01008=2100.071600,208.803900,-379.064600,0.389611,0.750575,-90.000210
C01009=2104.597400,208.803900,-377.906500,-2.245995,4.090919,-90.000210
C01010=2105.223500,208.803900,-378.895900,-0.366693,3.202834,-90.000210
C01011=2109.522500,208.803900,-378.143200,-3.758603,3.071054,-90.000210
C01012=2110.162200,208.803900,-377.230100,-6.783820,-0.492744,-90.000210
C01013=2113.905600,208.803900,-377.738500,-4.182592,3.913302,-90.000210
C01014=2115.676200,208.803900,-377.544600,-10.393454,3.752874,-90.000210
C01015=2116.867500,208.803900,-377.985800,-1.386558,3.111161,-90.000210
C01016=2119.696600,208.803900,-377.935100,-0.739116,3.197104,-90.000210
C01017=2121.655100,208.803900,-376.977600,5.563420,-4.555014,-90.000210
C01018=2124.496200,208.803900,-378.352800,0.504203,2.916355,-90.000210
C01019=2125.342000,208.803900,-378.091900,-4.537826,3.764333,-90.000210
C01020=2130.096500,208.803900,-377.169600,-2.824682,2.566851,-90.000210
C01021=2132.447100,208.803900,-376.804700,-1.059972,1.094349,-90.000210
C01022=2135.245400,208.803900,-377.232500,-0.131780,-5.895736,-90.000210
C01023=2136.828300,208.803900,-376.772800,-6.250970,3.626823,-90.000210
C01024=2139.609400,208.803900,-377.333200,-0.933921,6.056164,-90.000210
C01025=2140.815000,208.803900,-377.552500,-2.377775,0.395341,-90.000210
C01026=2144.185400,208.803900,-377.207200,-1.283425,1.180293,-90.000210
C01027=2145.974200,208.803900,-377.282500,-2.274642,-0.126051,-90.000210
C01028=2149.228400,208.803900,-377.060400,-4.039352,3.323155,-90.000210
C01029=2150.114300,208.803900,-377.167500,0.853707,1.764710,-90.000210
C01030=2151.355700,208.803900,-376.906800,2.039730,1.163104,-90.000210
C01031=2154.711000,208.803900,-377.071700,-4.045082,-1.117268,-90.000210
C01032=2155.831400,208.803900,-377.169000,1.695955,-2.108485,-90.000210
C01033=2158.437800,208.803900,-377.483700,-3.008028,2.830412,-90.000210
C01034=2159.759500,208.803900,-376.882100,-0.733386,0.355234,-90.000210
C01035=2160.644800,208.803900,-376.885400,-1.002676,5.437369,-90.000210
C01036=2163.605400,208.803900,-376.753000,-1.569904,1.237589,-90.000210
C01037=2165.435000,208.803900,-376.757800,-1.352180,0.555769,-90.000210
C01038=2165.872300,208.803900,-377.076400,15.171922,-0.074485,-90.000210
C01039=2169.376400,208.803900,-377.119700,1.833465,-2.836141,-90.000210
C01040=2170.477100,208.803900,-376.733400,-3.632552,4.417505,-90.000210
C01041=2171.900000,208.803900,-377.095500,-4.331561,4.411775,-90.000210
C01042=2174.172600,208.803900,-376.883100,5.574879,-0.423989,-90.000210
C01043=2175.393900,208.803900,-377.068800,1.713144,2.039730,-90.000210
C01044=2177.857700,208.803900,-376.746400,0.572958,4.480530,-90.000210
C01045=2180.118300,208.803900,-376.259400,-1.546986,1.495420,-90.000210
C01046=2183.652600,208.803900,-377.007200,3.804440,-0.154699,-90.000210
C01047=2185.084100,208.803900,-376.532100,-4.663876,2.045459,-90.000210
C01048=2186.051300,158.803900,-375.227800,0.383882,-0.750575,-90.000210
C01049=2184.581300,158.803900,-375.378500,-2.503826,6.520260,-90.000210
C01050=2180.434300,158.803900,-376.133500,1.501149,4.852953,-90.000210
C01051=2179.702400,158.803900,-376.823300,-1.558445,6.113460,-90.000210
C01052=2175.880900,158.803900,-376.616200,-1.203211,5.884277,-90.000210
C01053=2174.439200,158.803900,-377.104700,-1.970975,3.065324,-90.000210
C01054=2173.422800,158.803900,-377.056300,-0.939651,5.878547,-90.000210
C01055=2170.660300,158.803900,-376.721400,1.707414,3.558068,-90.000210
C01056=2170.235400,158.803900,-376.503100,0.991217,0.487014,-90.000210
C01057=2169.305700,158.803900,-377.176700,-0.956840,3.013758,-90.000210
C01058=2167.225300,158.803900,-376.867600,-0.756304,5.391533,-90.000210
C01059=2165.148000,158.803900,-376.924600,-1.907949,2.824682,-90.000210
C01060=2164.554400,158.803900,-377.230500,0.080214,2.446530,-90.000210
C01061=2160.888700,158.803900,-377.453700,0.137510,2.635606,-90.000210
C01062=2160.115800,158.803900,-377.533600,-2.652795,2.669983,-90.000210
C01063=2155.393400,158.803900,-377.509000,-0.378152,1.587093,-90.000210
C01064=2154.510800,158.803900,-378.041200,0.635983,3.071054,-90.000210
C01065=2149.754900,158.803900,-377.602500,-0.985487,0.578687,-90.000210
C01066=2148.910200,158.803900,-377.636800,-2.738738,4.898789,-90.000210
C01067=2145.138700,158.803900,-378.176500,-4.205510,5.374344,-90.000210
C01068=2143.685100,158.803900,-377.478100,0.372423,2.836141,-90.000210
C01069=2140.371300,158.803900,-378.907100,-1.604282,4.572203,-90.000210
C01070=2139.559900,158.803900,-377.848200,-1.953786,2.383504,-90.000210
C01071=2135.153900,158.803900,-379.008000,-4.136755,1.415206,-90.000210
C01072=2134.071900,158.803900,-378.324600,-0.979758,1.827735,-90.000210
C01073=2130.265600,158.803900,-379.200200,-4.039352,3.179916,-90.000210
C01074=2129.504100,158.803900,-378.851600,-1.667307,4.761279,-90.000210
C01075=2124.870800,158.803900,-378.184900,-0.275020,3.111161,-90.000210
C01076=2124.336100,158.803900,-379.532000,-1.524068,2.687172,-90.000210
C01077=2119.547300,158.803900,-378.739400,-0.389611,1.575634,-90.000210
C01078=2118.678100,158.803900,-379.070000,0.475555,3.689848,-90.000210
C01079=2114.948700,158.803900,-379.673000,-0.034377,3.202834,-90.000210
C01080=2114.156900,158.803900,-379.062400,-1.925138,5.385803,-90.000210
C01081=2109.806800,158.803900,-379.761800,-2.675713,3.082513,-90.000210
C01082=2108.644300,158.803900,-379.351600,-2.331938,1.461042,-90.000210
C01083=2105.025800,158.803900,-379.781900,-6.285347,2.773116,-90.000210
C01084=2104.038400,158.803900,-380.327600,-0.670361,-0.727656,-90.000210
C01085=2099.906900,158.803900,-379.049000,-0.710468,-0.653172,-90.000210
C01086=2099.307800,158.803900,-379.441900,-1.186023,1.529797,-90.000210
C01087=2094.144600,158.803900,-379.808100,-5.133702,2.457989,-90.000210
C01088=2093.296300,158.803900,-380.550100,-2.813223,1.323533,-90.000210
C01089=2089.469500,158.803900,-380.757100,-2.601228,1.420935,-90.000210
C01090=2087.431400,158.803900,-380.036200,-0.074485,1.736062,-90.000210
C01091=2085.451700,158.803900,-380.723100,-2.566851,2.251724,-90.000210
C01092=2084.030700,158.803900,-380.832400,0.985487,3.059595,-90.000210
C01093=2080.035300,158.803900,-379.737900,-4.148214,3.483583,-90.000210
C01094=2079.484800,158.803900,-381.390500,-1.512609,1.489690,-90.000210
C01095=2074.709300,158.803900,-380.984000,-1.317803,3.380451,-90.000210
C01096=2074.032800,158.803900,-381.188900,-4.755550,4.858682,-90.000210
C01097=2070.281400,158.803900,-379.963900,0.360963,0.979758,-90.000210
C01098=2068.312500,158.803900,-381.360900,-2.200158,-0.962569,-90.000210
C01099=2065.267200,158.803900,-380.813600,-1.260507,0.280749,-90.000210
C01100=2064.509300,158.803900,-381.262100,-6.354102,4.022164,-90.000210
C01101=2060.241500,158.803900,-381.026300,-2.022541,1.002676,-90.000210
C01102=2059.134200,158.803900,-380.368300,-1.403747,5.477477,-90.000210
C01103=2055.026500,158.803900,-381.956500,-3.076783,0.802141,-90.000210
C01104=2053.840800,158.803900,-380.488600,1.334992,-0.842248,-90.000210
C01105=2050.032000,158.803900,-380.980700,-3.380451,3.162727,-90.000210
C01106=2049.382600,158.803900,-381.344200,-2.331938,-3.122620,-90.000210
C01107=2046.013100,158.803900,-381.188900,1.403747,-1.466772,-90.000210
C01108=2044.577400,158.803900,-381.354600,-4.927437,-0.423989,-90.000210
C01109=2043.336900,158.803900,-381.945700,-7.454181,3.844547,-90.000210
C01110=2040.178900,158.803900,-380.743700,-2.853330,4.050812,-90.000210
C01111=2038.975600,158.803900,-381.913700,1.122997,-2.618417,-90.000210
C01112=2034.929000,158.803900,-380.462400,-4.262806,2.635606,-90.000210
C01113=2034.396900,158.803900,-381.111800,-5.047758,2.326209,-90.000210
C01114=2033.042600,158.803900,-381.957200,-1.993893,0.320856,-90.000210
C01115=2029.727300,158.803900,-381.029000,-1.134456,-0.624524,-90.000210
C01116=2029.341200,158.803900,-382.295000,-0.670361,-1.214671,-90.000210
C01117=2025.552800,158.803900,-382.046100,0.275020,0.343775,-90.000210
C01118=2024.557700,158.803900,-382.231500,0.194806,1.334992,-90.000210
C01119=2020.436600,158.803900,-380.874500,-4.102378,0.423989,-90.000210
C01120=2019.721000,158.803900,-381.449200,-2.022541,0.452637,-90.000210
C01121=2016.222800,158.803900,-381.350300,-6.841116,0.435448,-90.000210
C01122=2014.762800,158.803900,-382.372600,1.140186,-0.916732,-90.000210
C01123=2012.972600,158.803900,-381.143200,-0.727656,0.727656,-90.000210
C01124=2010.802800,158.803900,-382.149500,1.186023,-1.724603,-90.000210
C01125=2009.611900,158.803900,-380.843600,-1.489690,-0.372423,-90.000210
C01126=2005.829300,158.803900,-382.603100,-6.703606,0.286479,-90.000210
C01127=2004.633600,158.803900,-380.983500,-3.071054,-0.670361,-90.000210
C01128=2003.963700,158.803900,-382.004800,-1.111538,-0.309397,-90.000210
C01129=1999.793600,158.803900,-381.636100,-1.598552,-1.753251,-90.000210
C01130=1998.672900,158.803900,-380.959200,-5.402992,1.604282,-90.000210
C01131=1995.138800,158.803900,-381.995000,3.328885,0.080214,-90.000210
C01132=1994.325000,158.803900,-382.180600,0.739116,1.386558,-90.000210
C01133=1991.038000,158.803900,-381.239900,-0.859437,-0.767763,-90.000210
C01134=1990.264900,158.803900,-381.404200,-2.349127,-1.220400,-90.000210
C01135=1987.335000,158.803900,-381.891700,4.606581,-0.240642,-90.000210
C01136=1985.001100,158.803900,-381.232400,-5.609257,0.939651,-90.000210
C01137=1983.940900,158.803900,-382.412300,0.979758,0.263561,-90.000210
C01138=1979.773100,158.803900,-381.409800,-1.438124,2.314749,-90.000210
C01139=1977.450000,158.803900,-382.265700,-5.460288,1.764710,-90.000210
C01140=1974.887900,158.803900,-381.518000,-6.806739,2.320479,-90.000210
C01141=1973.704000,158.803900,-381.791900,1.415206,4.234158,-90.000210
C01142=1971.251300,158.803900,-381.745500,1.357910,0.091673,-90.000210
C01143=1969.658600,158.803900,-382.264700,0.280749,2.801764,-90.000210
C01144=1968.961400,158.803900,-381.733600,-3.856006,-5.150891,-90.000210
C01145=1965.016900,158.803900,-382.561100,-1.478231,-0.916732,-90.000210
C01146=1964.109300,158.803900,-382.767400,-5.529043,1.764710,-90.000210
C01147=1960.588200,158.803900,-381.399900,-3.260130,0.647442,-90.000210
C01148=1959.256600,158.803900,-381.765900,-1.936597,3.380451,-90.000210
C01149=1956.483200,158.803900,-381.654900,-2.039730,2.211617,-90.000210
C01150=1954.915600,158.803900,-382.719000,-1.804817,0.796411,-90.000210
C01151=1951.244200,158.803900,-381.753400,1.008406,6.302536,-90.000210
C01152=1949.542500,158.803900,-380.959800,-3.649741,0.813600,-90.000210
C01153=1948.564300,158.803900,-382.650300,3.592445,0.956840,-90.000210
C01154=1944.845300,158.803900,-382.989900,-4.870141,2.412152,-90.000210
C01155=1943.650800,158.803900,-382.854500,-0.137510,2.297561,-90.000210
C01156=1940.249700,158.803900,-382.312600,0.389611,0.550039,-90.000210
C01157=1939.985300,158.803900,-383.091300,-1.638659,5.666553,-90.000210
C01158=1936.858400,158.803900,-382.264100,-5.053488,1.426665,-90.000210
C01159=1935.151400,158.803900,-382.287200,0.349504,0.870896,-90.000210
C01160=1931.866900,158.803900,-382.106700,-3.603905,3.030947,-90.000210
C01161=1929.856100,158.803900,-383.067300,-2.876248,-1.306344,-90.000210
C01162=1928.280700,158.803900,-381.657200,-0.888085,-1.919409,-90.000210
C01163=1924.931800,158.803900,-383.328900,-2.177240,-0.263561,-90.000210
C01164=1924.145000,158.803900,-382.535200,-5.614986,2.578310,-90.000210
C01165=1920.513000,158.803900,-382.142900,-3.420558,-0.418259,-90.000210
C01166=1919.312200,158.803900,-382.391500,-1.781899,-2.217347,-90.000210
C01167=1914.493600,158.803900,-382.086100,-2.417882,1.804817,-90.000210
C01168=1914.330000,158.803900,-382.749200,2.475178,-1.289155,-90.000210
C01169=1911.180500,158.803900,-382.835200,-2.005352,2.830412,-90.000210
C01170=1909.902300,158.803900,-381.762700,-7.288023,-0.544310,-90.000210
C01171=1906.067500,158.803900,-382.842300,1.323533,-0.458366,-90.000210
C01172=1905.011400,158.803900,-382.641700,-3.586716,-1.592823,-90.000210
C01173=1900.583300,158.803900,-382.797500,-1.781899,-1.604282,-90.000210
C01174=1899.788500,158.803900,-382.172400,-1.930868,-0.825059,-90.000210
C01175=1895.760300,158.803900,-381.886400,-4.234158,0.550039,-90.000210
C01176=1894.594800,158.803900,-382.626400,-3.466395,-1.312073,-90.000210
C01177=1892.203800,158.803900,-382.091200,-3.964868,-1.375099,-90.000210
C01178=1890.022100,158.803900,-381.622200,-1.850654,-2.698631,-90.000210
C01179=1888.748500,158.803900,-381.651900,-4.159674,-4.503448,-90.000210
C01180=1885.598500,158.803900,-381.584100,1.174563,3.970598,-90.000210
C01181=1884.835900,158.803900,-382.372900,-4.847223,0.040107,-90.000210
C01182=1883.408600,158.803900,-381.827600,-4.606581,-2.177240,-90.000210
C01183=1879.477700,158.803900,-382.180900,-1.506879,-0.985487,-90.000210
C01184=1878.971200,158.803900,-381.181700,-0.876625,-2.400693,-90.000210
C01185=1874.971300,158.803900,-381.141900,-2.280372,-0.670361,-90.000210
C01186=1874.190200,158.803900,-382.209700,-0.252101,-2.492366,-90.000210
C01187=1870.334600,158.803900,-380.407600,-3.472124,-0.011459,-90.000210
C01188=1869.469500,158.803900,-381.574900,-4.698254,-0.292208,-90.000210
C01189=1865.393800,158.803900,-380.688300,-3.363262,-3.317426,-90.000210
C01190=1864.744400,158.803900,-380.585500,1.197482,0.383882,-90.000210
C01191=1862.140000,158.803900,-382.096500,-5.912924,-4.612310,-90.000210
C01192=1860.194400,158.803900,-380.808300,-2.280372,-2.755927,-90.000210
C01193=1859.245000,158.803900,-381.117900,-0.956840,-0.257831,-90.000210
C01194=1855.289000,158.803900,-380.403700,0.189076,-4.658147,-90.000210
C01195=1854.730000,158.803900,-380.374900,-0.343775,-1.065701,-90.000210
C01196=1850.109200,158.803900,-380.039200,-5.506124,-1.862113,-90.000210
C01197=1849.392200,158.803900,-380.126300,-3.575257,-5.592068,-90.000210
C01198=1845.224000,158.803900,-379.567600,-3.489313,0.865166,-90.000210
C01199=1844.348600,158.803900,-379.823300,-5.861358,-1.346451,-90.000210
C01200=1840.144500,158.803900,-379.377400,-0.429718,-2.767386,-90.000210
C01201=1839.522700,158.803900,-380.278200,-4.205510,-3.924761,-90.000210
C01202=1835.275500,158.803900,-379.806800,-4.331561,-0.802141,-90.000210
C01203=1834.424500,158.803900,-380.477800,-1.094349,-3.901843,-90.000210
C01204=1830.269300,158.803900,-379.575500,2.578310,-1.357910,-90.000210
C01205=1828.414400,158.803900,-378.766800,-2.956462,-0.876625,-90.000210
C01206=1824.701500,158.803900,-378.747700,-2.475178,-0.784952,-90.000210
C01207=1823.852600,158.803900,-379.628700,-2.813223,0.000000,-90.000210
C01208=1819.681600,158.803900,-379.287300,-1.695955,-3.598175,-90.000210
C01209=1818.352100,158.803900,-379.128900,0.040107,-1.610011,-90.000210
C01210=1815.253300,158.803900,-378.511700,0.487014,-2.377775,-90.000210
C01211=1814.405100,158.803900,-378.620900,-3.340344,-0.996947,-90.000210
C01212=1810.294700,158.803900,-378.646300,-0.750575,-3.380451,-90.000210
C01213=1808.202800,158.803900,-378.307100,-1.558445,-0.487014,-90.000210
C01214=1805.361300,158.803900,-378.314600,-0.355234,-4.222699,-90.000210
C01215=1803.949600,158.803900,-378.205400,0.630254,-0.527121,-90.000210
C01216=1800.699800,158.803900,-378.463900,-2.389234,-6.886953,-90.000210
C01217=1799.347800,158.803900,-377.779000,-0.051566,-2.647065,-90.000210
C01218=1795.852200,158.803900,-377.554000,0.303668,3.294507,-90.000210
C01219=1794.744200,108.803900,-377.373000,-1.827735,-6.365561,-90.000210
C01220=1795.283000,108.803900,-377.674900,-0.676090,-6.004598,-90.000210
C01221=1798.437200,108.803900,-378.634900,-4.113837,-7.580232,-90.000210
C01222=1799.550600,108.803900,-378.136900,-4.778468,-1.988164,-90.000210
C01223=1804.214700,108.803900,-378.939500,1.873572,-6.715065,-90.000210
C01224=1805.330300,108.803900,-378.791900,-0.865166,-4.010705,-90.000210
C01225=1809.117600,108.803900,-378.677700,-4.153944,-2.876248,-90.000210
C01226=1810.050200,108.803900,-379.328000,1.667307,-2.967921,-90.000210
C01227=1812.965400,108.803900,-379.523200,0.206265,-3.397640,-90.000210
C01228=1814.493100,108.803900,-379.691100,-1.907949,-6.268158,-90.000210
C01229=1818.922600,108.803900,-379.770100,-1.587093,-4.285724,-90.000210
C01230=1819.903900,108.803900,-380.055300,0.704738,-3.792981,-90.000210
C01231=1823.323000,108.803900,-379.996000,0.343775,-0.492744,-90.000210
C01232=1824.695300,108.803900,-379.868300,-1.770440,-3.689848,-90.000210
C01233=1829.240200,108.803900,-380.232100,0.338045,-1.632930,-90.000210
C01234=1830.010700,108.803900,-380.649600,0.538580,-0.366693,-90.000210
C01235=1832.538900,108.803900,-380.599300,-1.827735,-4.216969,-90.000210
C01236=1834.830000,108.803900,-380.317700,-1.804817,-4.314372,-90.000210
C01237=1839.193700,108.803900,-380.576900,-2.400693,-3.454936,-90.000210
C01238=1840.213800,108.803900,-380.897200,-1.953786,-2.584040,-90.000210
C01239=1843.785200,108.803900,-381.601100,-0.492744,-4.543555,-90.000210
C01240=1845.473900,108.803900,-381.963100,0.601606,-4.789927,-90.000210
C01241=1845.654800,108.803900,-381.932200,-0.527121,-2.515285,-90.000210
C01242=1849.452600,108.803900,-381.793200,-3.523690,1.048513,-90.000210
C01243=1850.223700,108.803900,-381.879000,-0.658901,-0.561499,-90.000210
C01244=1851.727200,108.803900,-382.056000,1.896490,-3.151268,-90.000210
C01245=1854.851200,108.803900,-382.035500,-2.469448,-1.100079,-90.000210
C01246=1855.709000,108.803900,-381.449800,0.464096,-3.374721,-90.000210
C01247=1859.761000,108.803900,-382.440600,0.171887,-1.816276,-90.000210
C01248=1860.563800,108.803900,-382.517100,-3.093972,-2.509555,-90.000210
C01249=1861.767400,108.803900,-381.993700,-1.277696,-5.551961,-90.000210
C01250=1864.201700,108.803900,-382.523700,-0.057296,-1.936597,-90.000210
C01251=1866.076400,108.803900,-382.567700,-2.904896,0.784952,-90.000210
C01252=1869.525700,108.803900,-382.551200,-1.890761,-2.091296,-90.000210
C01253=1870.289800,108.803900,-382.429900,-1.369369,-2.853330,-90.000210
C01254=1875.008800,108.803900,-382.747800,-0.956840,0.189076,-90.000210
C01255=1876.033500,108.803900,-382.632200,-5.311319,0.538580,-90.000210
C01256=1879.817000,108.803900,-382.586100,-1.569904,-1.552716,-90.000210
C01257=1880.355300,108.803900,-382.620300,4.073730,-4.761279,-90.000210
C01258=1884.434200,108.803900,-383.154200,-2.326209,-2.990840,-90.000210
C01259=1885.347400,108.803900,-383.047300,-2.251724,-2.704361,-90.000210
C01260=1889.287700,108.803900,-383.436700,0.727656,-0.372423,-90.000210
C01261=1890.720900,108.803900,-382.878700,-3.615364,1.839195,-90.000210
C01262=1894.258800,108.803900,-383.326500,0.446907,-1.489690,-90.000210
C01263=1896.162500,108.803900,-382.987500,-0.836518,-2.291831,-90.000210
C01264=1899.897200,108.803900,-383.389000,-0.091673,-1.186023,-90.000210
C01265=1900.916100,108.803900,-383.403800,-2.566851,-0.303668,-90.000210
C01266=1905.062700,108.803900,-383.932200,-2.045459,-1.254778,-90.000210
C01267=1905.704900,108.803900,-383.234100,0.074485,2.286102,-90.000210
C01268=1908.888300,108.803900,-383.727500,-1.386558,0.223454,-90.000210
C01269=1909.936300,108.803900,-383.142000,-5.282671,-0.143239,-90.000210
C01270=1914.697500,108.803900,-383.117700,-4.801386,-0.051566,-90.000210
C01271=1916.137100,108.803900,-383.399200,-0.223454,3.586716,-90.000210
C01272=1919.285400,108.803900,-383.089400,-2.996569,0.979758,-90.000210
C01273=1919.909800,108.803900,-383.805600,0.613065,-1.569904,-90.000210
C01274=1924.508500,108.803900,-383.980700,-0.567228,-2.492366,-90.000210
C01275=1925.664800,108.803900,-383.772500,-5.185268,7.184891,-90.000210
C01276=1929.305000,108.803900,-383.905700,0.893814,0.406800,-90.000210
C01277=1930.380700,108.803900,-383.246600,-2.750197,-2.922085,-90.000210
C01278=1934.724900,108.803900,-383.324800,1.942327,0.727656,-90.000210
C01279=1936.137200,108.803900,-383.827200,-2.062648,0.383882,-90.000210
C01280=1939.690500,108.803900,-383.432000,0.670361,3.048135,-90.000210
C01281=1940.791900,108.803900,-384.389500,1.690225,-2.624147,-90.000210
C01282=1944.547300,108.803900,-383.113900,0.555769,-0.045837,-90.000210
C01283=1945.223700,108.803900,-383.374300,6.766632,6.193674,-90.000210
C01284=1949.590000,108.803900,-383.510400,0.865166,0.509932,-90.000210
C01285=1950.926900,108.803900,-383.959800,2.268913,3.340344,-90.000210
C01286=1955.180000,108.803900,-383.004400,1.306344,-2.406423,-90.000210
C01287=1956.475000,108.803900,-383.052800,-3.947679,1.231859,-90.000210
C01288=1959.975700,108.803900,-383.156400,0.561499,1.191752,-90.000210
C01289=1960.732000,108.803900,-383.011000,-5.190998,0.429718,-90.000210
C01290=1964.501800,108.803900,-383.214900,-0.183346,5.391533,-90.000210
C01291=1966.277700,108.803900,-383.011900,1.254778,-0.836518,-90.000210
C01292=1969.836300,108.803900,-383.713100,0.446907,4.136755,-90.000210
C01293=1970.819000,108.803900,-383.013000,-0.406800,-0.280749,-90.000210
C01294=1974.872100,108.803900,-383.569500,-0.257831,2.137133,-90.000210
C01295=1975.784200,108.803900,-383.326000,-1.415206,-0.515662,-90.000210
C01296=1980.213900,108.803900,-383.311600,-2.738738,1.483961,-90.000210
C01297=1980.915100,108.803900,-383.012500,-1.163104,0.114592,-90.000210
C01298=1984.723200,108.803900,-382.898300,-4.428964,0.068755,-90.000210
C01299=1985.767600,108.803900,-383.269300,0.332316,1.140186,-90.000210
C01300=1990.375700,108.803900,-382.755000,3.632552,-1.982434,-90.000210
C01301=1991.153100,108.803900,-382.934600,-2.572581,1.231859,-90.000210
C01302=1994.951400,108.803900,-382.911100,-1.988164,1.117268,-90.000210
C01303=1995.784400,108.803900,-382.933600,-0.326586,1.031324,-90.000210
C01304=1999.864000,108.803900,-382.796200,-2.635606,1.168834,-90.000210
C01305=2000.574700,108.803900,-382.692100,-0.733386,-1.461042,-90.000210
C01306=2004.866300,108.803900,-383.199200,-0.544310,2.056918,-90.000210
C01307=2007.056000,108.803900,-383.284800,0.979758,-1.357910,-90.000210
C01308=2009.897700,108.803900,-382.958100,0.779223,2.440800,-90.000210
C01309=2010.997300,108.803900,-382.499300,3.747144,1.970975,-90.000210
C01310=2014.605500,108.803900,-383.059400,1.277696,0.911003,-90.000210
C01311=2015.715000,108.803900,-382.609500,4.222699,2.578310,-90.000210
C01312=2019.736500,108.803900,-382.900200,-5.362885,1.340721,-90.000210
C01313=2020.984000,108.803900,-383.145400,-0.699009,3.305966,-90.000210
C01314=2024.713700,108.803900,-382.436400,-2.349127,1.982434,-90.000210
C01315=2025.539800,108.803900,-382.856200,-4.159674,2.326209,-90.000210
C01316=2029.502500,108.803900,-382.819500,-6.222322,-1.535527,-90.000210
C01317=2031.463900,108.803900,-382.252500,-4.807116,2.601228,-90.000210
C01318=2034.505800,108.803900,-382.390200,-7.935465,3.317426,-90.000210
C01319=2035.972500,108.803900,-382.159400,-4.004975,0.057296,-90.000210
C01320=2039.787700,108.803900,-382.187500,-4.692524,1.667307,-90.000210
C01321=2040.832500,108.803900,-383.110900,1.128727,-1.420935,-90.000210
C01322=2044.710700,108.803900,-382.573400,-1.008406,-0.280749,-90.000210
C01323=2045.413900,108.803900,-382.211100,-3.924761,5.311319,-90.000210
C01324=2049.724600,108.803900,-382.574200,3.552338,-0.750575,-90.000210
C01325=2050.256300,108.803900,-382.121200,0.555769,0.962569,-90.000210
C01326=2051.382800,108.803900,-381.752000,0.234913,2.939273,-90.000210
C01327=2054.010400,108.803900,-382.504400,-0.286479,1.776169,-90.000210
C01328=2055.568300,108.803900,-382.106800,-0.572958,0.836518,-90.000210
C01329=2059.213500,108.803900,-382.574900,-1.472502,0.160428,-90.000210
C01330=2060.480700,108.803900,-382.559900,1.375099,1.260507,-90.000210
C01331=2063.614100,108.803900,-382.682200,-1.134456,-3.323155,-90.000210
C01332=2065.104300,108.803900,-382.001600,2.074107,2.584040,-90.000210
C01333=2066.757500,108.803900,-382.084600,-0.389611,-0.355234,-90.000210
C01334=2069.094400,108.803900,-382.215300,-1.885031,7.127595,-90.000210
C01335=2070.547700,108.803900,-382.302200,3.168457,-0.137510,-90.000210
C01336=2072.932300,108.803900,-382.198200,-5.345696,6.067623,-90.000210
C01337=2074.436100,108.803900,-381.761100,-3.827358,5.712389,-90.000210
C01338=2076.512900,108.803900,-382.087600,-2.578310,-0.842248,-90.000210
C01339=2079.098400,108.803900,-382.350700,-7.534395,11.000790,-90.000210
C01340=2080.360800,108.803900,-381.448500,-4.102378,5.311319,-90.000210
C01341=2081.878800,108.803900,-382.094200,-5.998868,1.655848,-90.000210
C01342=2084.796700,108.803900,-381.398400,-4.566474,1.529797,-90.000210
C01343=2085.871700,108.803900,-381.549900,-0.911003,4.858682,-90.000210
C01344=2089.136500,108.803900,-381.599100,-1.793358,1.896490,-90.000210
C01345=2090.023600,108.803900,-381.861000,1.054242,-0.721927,-90.000210
C01346=2093.346200,108.803900,-381.946000,-1.850654,-6.136378,-90.000210
C01347=2094.329100,108.803900,-381.454500,-3.351803,6.726525,-90.000210
C01348=2098.156600,108.803900,-381.345400,0.378152,0.670361,-90.000210
C01349=2100.038800,108.803900,-380.948000,-2.062648,0.315127,-90.000210
C01350=2103.365500,108.803900,-380.867900,-1.993893,2.910626,-90.000210
C01351=2105.270500,108.803900,-380.870600,-1.999623,4.406045,-90.000210
C01352=2108.636100,108.803900,-380.785300,0.000000,4.807116,-90.000210
C01353=2110.171600,108.803900,-380.810600,-1.770440,2.538203,-90.000210
C01354=2114.318200,108.803900,-380.633500,-2.211617,2.635606,-90.000210
C01355=2114.968600,108.803900,-380.419500,1.375099,3.225752,-90.000210
C01356=2118.593700,108.803900,-380.570400,-2.309020,5.362885,-90.000210
C01357=2119.933100,108.803900,-380.360500,0.487014,3.128350,-90.000210
C01358=2123.489900,108.803900,-379.750700,-4.864412,4.343020,-90.000210
C01359=2124.467200,108.803900,-379.731800,1.094349,4.348750,-90.000210
C01360=2128.885100,108.803900,-379.930700,0.435448,2.658524,-90.000210
C01361=2129.833500,108.803900,-379.787800,-0.670361,3.368992,-90.000210
C01362=2134.538400,108.803900,-379.118800,-0.830789,2.389234,-90.000210
C01363=2135.914500,108.803900,-379.359300,-1.718873,3.248671,-90.000210
C01364=2139.422800,108.803900,-379.144000,-1.415206,4.938896,-90.000210
